    R361_2_O_RB_이상_리셋 AT %MW94020.10 : BOOL; (* R361_2_O_RB_이상_리셋 *)
    R361_2_O_RB_작업완료_리셋 AT %MW94020.8 : BOOL; (* R361_2_O_RB_작업완료_리셋 *)
    R363_1_I_RB_0_5_COMM_CHK AT %MW84033.14 : BOOL; (* R363_1_I_RB_0_5_COMM_CHK *)
    R363_1_I_RB_10차_간섭무 AT %MW84031.9 : BOOL; (* R363_1_I_RB_10차_간섭무 *)
    R363_1_I_RB_11차_간섭무 AT %MW84031.10 : BOOL; (* R363_1_I_RB_11차_간섭무 *)
    R363_1_I_RB_12차_간섭무 AT %MW84031.11 : BOOL; (* R363_1_I_RB_12차_간섭무 *)
    R363_1_I_RB_1차_간섭무 AT %MW84031.0 : BOOL; (* R363_1_I_RB_1차_간섭무 *)
    R363_1_I_RB_1차_작업완료 AT %MW84030.9 : BOOL; (* R363_1_I_RB_1차_작업완료 *)
    R363_1_I_RB_2차_간섭무 AT %MW84031.1 : BOOL; (* R363_1_I_RB_2차_간섭무 *)
    R363_1_I_RB_2차_작업완료 AT %MW84030.10 : BOOL; (* R363_1_I_RB_2차_작업완료 *)
    R363_1_I_RB_3차_간섭무 AT %MW84031.2 : BOOL; (* R363_1_I_RB_3차_간섭무 *)
    R363_1_I_RB_3차_작업완료 AT %MW84030.11 : BOOL; (* R363_1_I_RB_3차_작업완료 *)
    R363_1_I_RB_4차_간섭무 AT %MW84031.3 : BOOL; (* R363_1_I_RB_4차_간섭무 *)
    R363_1_I_RB_4차_작업완료 AT %MW84030.12 : BOOL; (* R363_1_I_RB_4차_작업완료 *)
    R363_1_I_RB_5차_간섭무 AT %MW84031.4 : BOOL; (* R363_1_I_RB_5차_간섭무 *)
    R363_1_I_RB_5차_작업완료 AT %MW84030.13 : BOOL; (* R363_1_I_RB_5차_작업완료 *)
    R363_1_I_RB_6차_간섭무 AT %MW84031.5 : BOOL; (* R363_1_I_RB_6차_간섭무 *)
    R363_1_I_RB_6차_작업완료 AT %MW84030.14 : BOOL; (* R363_1_I_RB_6차_작업완료 *)
    R363_1_I_RB_7차_간섭무 AT %MW84031.6 : BOOL; (* R363_1_I_RB_7차_간섭무 *)
    R363_1_I_RB_7차_작업완료 AT %MW84030.15 : BOOL; (* R363_1_I_RB_7차_작업완료 *)
    R363_1_I_RB_8차_간섭무 AT %MW84031.7 : BOOL; (* R363_1_I_RB_8차_간섭무 *)
    R363_1_I_RB_9차_간섭무 AT %MW84031.8 : BOOL; (* R363_1_I_RB_9차_간섭무 *)
    R363_1_I_RB_AB_NORMAL_선택 AT %MW84030.6 : BOOL; (* R363_1_I_RB_AB_NORMAL_선택 *)
    R363_1_I_RB_GUN1_FIXED_TIP AT %MW84037 : WORD; (* R363_1_I_RB_GUN1_FIXED_TIP *)
    R363_1_I_RB_GUN1_MOVING_TIP AT %MW84036 : WORD; (* R363_1_I_RB_GUN1_MOVING_TIP *)
    R363_1_I_RB_GUN2_FIXED_TIP AT %MW84039 : WORD; (* R363_1_I_RB_GUN2_FIXED_TIP *)
    R363_1_I_RB_GUN2_MOVING_TIP AT %MW84038 : WORD; (* R363_1_I_RB_GUN2_MOVING_TIP *)
    R363_1_I_RB_INPUT AT %MW84030 : ARRAY[0..3] OF WORD; (* R363_1_I_RB_INPUT *)
    R363_1_I_RB_LS_이상 AT %MW84032.11 : BOOL; (* R363_1_I_RB_LS_이상 *)
    R363_1_I_RB_MOTOR_MC_ON AT %MW84033.15 : BOOL; (* R363_1_I_RB_MOTOR_MC_ON *)
    R363_1_I_RB_PLT_UNLOAD_완료 AT %MW84033.11 : BOOL; (* R363_1_I_RB_PLT_UNLOAD_완료 *)
    R363_1_I_RB_PLT_최종UNLOAD_완료 AT %MW84033.12 : BOOL; (* R363_1_I_RB_PLT_최종UNLOAD_완료 *)
    R363_1_I_RB_PROG_ECHO_1 AT %MW84032.0 : BOOL; (* R363_1_I_RB_PROG_ECHO_1 *)
    R363_1_I_RB_PROG_ECHO_128 AT %MW84032.7 : BOOL; (* R363_1_I_RB_PROG_ECHO_128 *)
    R363_1_I_RB_PROG_ECHO_16 AT %MW84032.4 : BOOL; (* R363_1_I_RB_PROG_ECHO_16 *)
    R363_1_I_RB_PROG_ECHO_2 AT %MW84032.1 : BOOL; (* R363_1_I_RB_PROG_ECHO_2 *)
    R363_1_I_RB_PROG_ECHO_32 AT %MW84032.5 : BOOL; (* R363_1_I_RB_PROG_ECHO_32 *)
    R363_1_I_RB_PROG_ECHO_4 AT %MW84032.2 : BOOL; (* R363_1_I_RB_PROG_ECHO_4 *)
    R363_1_I_RB_PROG_ECHO_64 AT %MW84032.6 : BOOL; (* R363_1_I_RB_PROG_ECHO_64 *)
    R363_1_I_RB_PROG_ECHO_8 AT %MW84032.3 : BOOL; (* R363_1_I_RB_PROG_ECHO_8 *)
    R363_1_I_RB_SP3_8 AT %MW84033.8 : BOOL; (* R363_1_I_RB_SP3_8 *)
    R363_1_I_RB_SP3_9 AT %MW84033.9 : BOOL; (* R363_1_I_RB_SP3_9 *)
    R363_1_I_RB_SPARE_WORD_4 AT %MW84034 : WORD; (* R363_1_I_RB_SPARE_WORD_4 *)
    R363_1_I_RB_SP_1_12 AT %MW84031.12 : BOOL; (* R363_1_I_RB_SP_1_12 *)
    R363_1_I_RB_SP_1_13 AT %MW84031.13 : BOOL; (* R363_1_I_RB_SP_1_13 *)
    R363_1_I_RB_SP_1_14 AT %MW84031.14 : BOOL; (* R363_1_I_RB_SP_1_14 *)
    R363_1_I_RB_SP_1_15 AT %MW84031.15 : BOOL; (* R363_1_I_RB_SP_1_15 *)
    R363_1_I_RB_TC_이상 AT %MW84032.8 : BOOL; (* R363_1_I_RB_TC_이상 *)
    R363_1_I_RB_TIP_CHANGE AT %MW84033.13 : BOOL; (* R363_1_I_RB_TIP_CHANGE *)
    R363_1_I_RB_TIP_DRESSING AT %MW84030.7 : BOOL; (* R363_1_I_RB_TIP_DRESSING *)
    R363_1_I_RB__PLT_카운터리셋완료 AT %MW84033.10 : BOOL; (* R363_1_I_RB__PLT_카운터리셋완료 *)
    R363_1_I_RB_공기압_이상 AT %MW84032.9 : BOOL; (* R363_1_I_RB_공기압_이상 *)
    R363_1_I_RB_냉각수_이상 AT %MW84032.10 : BOOL; (* R363_1_I_RB_냉각수_이상 *)
    R363_1_I_RB_비상정지_NC AT %MW84030.8 : BOOL; (* R363_1_I_RB_비상정지_NC *)
    R363_1_I_RB_비전이상 AT %MW84032.14 : BOOL; (* R363_1_I_RB_비전이상 *)
    R363_1_I_RB_상호인터록_INT1 AT %MW84033.0 : BOOL; (* R363_1_I_RB_상호인터록_INT1 *)
    R363_1_I_RB_상호인터록_INT2 AT %MW84033.1 : BOOL; (* R363_1_I_RB_상호인터록_INT2 *)
    R363_1_I_RB_상호인터록_INT3 AT %MW84033.2 : BOOL; (* R363_1_I_RB_상호인터록_INT3 *)
    R363_1_I_RB_상호인터록_INT4 AT %MW84033.3 : BOOL; (* R363_1_I_RB_상호인터록_INT4 *)
    R363_1_I_RB_상호인터록_INT5 AT %MW84033.4 : BOOL; (* R363_1_I_RB_상호인터록_INT5 *)
    R363_1_I_RB_상호인터록_INT6 AT %MW84033.5 : BOOL; (* R363_1_I_RB_상호인터록_INT6 *)
    R363_1_I_RB_상호인터록_INT7 AT %MW84033.6 : BOOL; (* R363_1_I_RB_상호인터록_INT7 *)
    R363_1_I_RB_상호인터록_INT8 AT %MW84033.7 : BOOL; (* R363_1_I_RB_상호인터록_INT8 *)
    R363_1_I_RB_실러이상 AT %MW84032.13 : BOOL; (* R363_1_I_RB_실러이상 *)
    R363_1_I_RB_용접카운터이상 AT %MW84032.15 : BOOL; (* R363_1_I_RB_용접카운터이상 *)
    R363_1_I_RB_용접타점수 AT %MW84035 : WORD; (* R363_1_I_RB_용접타점수 *)
    R363_1_I_RB_운전준비 AT %MW84030.3 : BOOL; (* R363_1_I_RB_운전준비 *)
    R363_1_I_RB_원위치 AT %MW84030.0 : BOOL; (* R363_1_I_RB_원위치 *)
    R363_1_I_RB_이상리셋 AT %MW84030.2 : BOOL; (* R363_1_I_RB_이상리셋 *)
    R363_1_I_RB_자동 AT %MW84030.4 : BOOL; (* R363_1_I_RB_자동 *)
    R363_1_I_RB_자동기동 AT %MW84030.5 : BOOL; (* R363_1_I_RB_자동기동 *)
    R363_1_I_RB_최종_작업완료 AT %MW84030.1 : BOOL; (* R363_1_I_RB_최종_작업완료 *)
    R363_1_I_RB_통신이상 AT %MW84032.12 : BOOL; (* R363_1_I_RB_통신이상 *)
    R363_1_M_I_RB_1차_작업완료 AT %MW20031.2 : BOOL; (* R363_1_M_I_RB_1차_작업완료 *)
    R363_1_M_I_RB_2차_작업완료 AT %MW20031.3 : BOOL; (* R363_1_M_I_RB_2차_작업완료 *)
    R363_1_M_I_RB_3차_작업완료 AT %MW20031.4 : BOOL; (* R363_1_M_I_RB_3차_작업완료 *)
    R363_1_M_I_RB_4차_작업완료 AT %MW20031.5 : BOOL; (* R363_1_M_I_RB_4차_작업완료 *)
    R363_1_M_I_RB_5차_작업완료 AT %MW20031.6 : BOOL; (* R363_1_M_I_RB_5차_작업완료 *)
    R363_1_M_I_RB_6차_작업완료 AT %MW20031.7 : BOOL; (* R363_1_M_I_RB_6차_작업완료 *)
    R363_1_M_I_RB_7차_작업완료 AT %MW20031.8 : BOOL; (* R363_1_M_I_RB_7차_작업완료 *)
    R363_1_M_I_RB_PAUSE_보조 AT %MW20030.5 : BOOL; (* R363_1_M_I_RB_PAUSE_보조 *)
    R363_1_M_I_RB_PLC_RUN_CHK_이상 AT %MW20030.7 : BOOL; (* R363_1_M_I_RB_PLC_RUN_CHK_이상 *)
    R363_1_M_I_RB_간섭무_1 AT %MW20032.0 : BOOL; (* R363_1_M_I_RB_간섭무_1 *)
    R363_1_M_I_RB_간섭무_10 AT %MW20032.9 : BOOL; (* R363_1_M_I_RB_간섭무_10 *)
    R363_1_M_I_RB_간섭무_11 AT %MW20032.10 : BOOL; (* R363_1_M_I_RB_간섭무_11 *)
    R363_1_M_I_RB_간섭무_12 AT %MW20032.11 : BOOL; (* R363_1_M_I_RB_간섭무_12 *)
    R363_1_M_I_RB_간섭무_2 AT %MW20032.1 : BOOL; (* R363_1_M_I_RB_간섭무_2 *)
    R363_1_M_I_RB_간섭무_3 AT %MW20032.2 : BOOL; (* R363_1_M_I_RB_간섭무_3 *)
    R363_1_M_I_RB_간섭무_4 AT %MW20032.3 : BOOL; (* R363_1_M_I_RB_간섭무_4 *)
    R363_1_M_I_RB_간섭무_5 AT %MW20032.4 : BOOL; (* R363_1_M_I_RB_간섭무_5 *)
    R363_1_M_I_RB_간섭무_6 AT %MW20032.5 : BOOL; (* R363_1_M_I_RB_간섭무_6 *)
    R363_1_M_I_RB_간섭무_7 AT %MW20032.6 : BOOL; (* R363_1_M_I_RB_간섭무_7 *)
    R363_1_M_I_RB_간섭무_8 AT %MW20032.7 : BOOL; (* R363_1_M_I_RB_간섭무_8 *)
    R363_1_M_I_RB_간섭무_9 AT %MW20032.8 : BOOL; (* R363_1_M_I_RB_간섭무_9 *)
    R363_1_M_I_RB_비상정지 AT %MW20030.4 : BOOL; (* R363_1_M_I_RB_비상정지 *)
    R363_1_M_I_RB_운전준비 AT %MW20030.0 : BOOL; (* R363_1_M_I_RB_운전준비 *)
    R363_1_M_I_RB_원위치 AT %MW20030.3 : BOOL; (* R363_1_M_I_RB_원위치 *)
    R363_1_M_I_RB_이상 AT %MW20030.2 : BOOL; (* R363_1_M_I_RB_이상 *)
    R363_1_M_I_RB_자동 AT %MW20030.1 : BOOL; (* R363_1_M_I_RB_자동 *)
    R363_1_M_I_RB_최종작업완료 AT %MW20031.0 : BOOL; (* R363_1_M_I_RB_최종작업완료 *)
    R363_1_M_I_RB_프로그램_이상 AT %MW20030.6 : BOOL; (* R363_1_M_I_RB_프로그램_이상 *)
    R363_1_M_O_RB_1_CYCLE_SET AT %MW21030.3 : BOOL; (* R363_1_M_O_RB_1_CYCLE_SET *)
    R363_1_M_O_RB_1_CYCLE_리셋 AT %MW21030.4 : BOOL; (* R363_1_M_O_RB_1_CYCLE_리셋 *)
    R363_1_M_O_RB_1차_작업완료_리셋 AT %MW21032.0 : BOOL; (* R363_1_M_O_RB_1차_작업완료_리셋 *)
    R363_1_M_O_RB_2차_작업완료_리셋 AT %MW21032.1 : BOOL; (* R363_1_M_O_RB_2차_작업완료_리셋 *)
    R363_1_M_O_RB_2차_진입OK AT %MW21031.8 : BOOL; (* R363_1_M_O_RB_2차_진입OK *)
    R363_1_M_O_RB_3차_작업완료_리셋 AT %MW21032.2 : BOOL; (* R363_1_M_O_RB_3차_작업완료_리셋 *)
    R363_1_M_O_RB_3차_진입OK AT %MW21031.9 : BOOL; (* R363_1_M_O_RB_3차_진입OK *)
    R363_1_M_O_RB_4차_작업완료_리셋 AT %MW21032.3 : BOOL; (* R363_1_M_O_RB_4차_작업완료_리셋 *)
    R363_1_M_O_RB_4차_진입OK AT %MW21031.10 : BOOL; (* R363_1_M_O_RB_4차_진입OK *)
    R363_1_M_O_RB_5차_작업완료_리셋 AT %MW21032.4 : BOOL; (* R363_1_M_O_RB_5차_작업완료_리셋 *)
    R363_1_M_O_RB_5차_진입OK AT %MW21031.11 : BOOL; (* R363_1_M_O_RB_5차_진입OK *)
    R363_1_M_O_RB_6차_작업완료_리셋 AT %MW21032.5 : BOOL; (* R363_1_M_O_RB_6차_작업완료_리셋 *)
    R363_1_M_O_RB_6차_진입OK AT %MW21031.12 : BOOL; (* R363_1_M_O_RB_6차_진입OK *)
    R363_1_M_O_RB_7차_작업완료_리셋 AT %MW21032.6 : BOOL; (* R363_1_M_O_RB_7차_작업완료_리셋 *)
    R363_1_M_O_RB_7차_진입OK AT %MW21031.13 : BOOL; (* R363_1_M_O_RB_7차_진입OK *)
    R363_1_M_O_RB_ATD_OK AT %MW21030.6 : BOOL; (* R363_1_M_O_RB_ATD_OK *)
    R363_1_M_O_RB_PLT_10_진입OK AT %MW21033.10 : BOOL; (* R363_1_M_O_RB_PLT_10_진입OK *)
    R363_1_M_O_RB_PLT_11_진입OK AT %MW21033.11 : BOOL; (* R363_1_M_O_RB_PLT_11_진입OK *)
    R363_1_M_O_RB_PLT_12_진입OK AT %MW21033.12 : BOOL; (* R363_1_M_O_RB_PLT_12_진입OK *)
    R363_1_M_O_RB_PLT_1_진입OK AT %MW21033.1 : BOOL; (* R363_1_M_O_RB_PLT_1_진입OK *)
    R363_1_M_O_RB_PLT_2_진입OK AT %MW21033.2 : BOOL; (* R363_1_M_O_RB_PLT_2_진입OK *)
    R363_1_M_O_RB_PLT_3_진입OK AT %MW21033.3 : BOOL; (* R363_1_M_O_RB_PLT_3_진입OK *)
    R363_1_M_O_RB_PLT_4_진입OK AT %MW21033.4 : BOOL; (* R363_1_M_O_RB_PLT_4_진입OK *)
    R363_1_M_O_RB_PLT_5_진입OK AT %MW21033.5 : BOOL; (* R363_1_M_O_RB_PLT_5_진입OK *)
    R363_1_M_O_RB_PLT_6_진입OK AT %MW21033.6 : BOOL; (* R363_1_M_O_RB_PLT_6_진입OK *)
    R363_1_M_O_RB_PLT_7_진입OK AT %MW21033.7 : BOOL; (* R363_1_M_O_RB_PLT_7_진입OK *)
    R363_1_M_O_RB_PLT_8_진입OK AT %MW21033.8 : BOOL; (* R363_1_M_O_RB_PLT_8_진입OK *)
    R363_1_M_O_RB_PLT_9_진입OK AT %MW21033.9 : BOOL; (* R363_1_M_O_RB_PLT_9_진입OK *)
    R363_1_M_O_RB_PLT_카운터리셋_보조 AT %MW21030.10 : BOOL; (* R363_1_M_O_RB_PLT_카운터리셋_보조 *)
    R363_1_M_O_RB_PROG_NO AT %MW21034 : WORD;
    R363_1_M_O_RB_RESTART_OK AT %MW21030.2 : BOOL; (* R363_1_M_O_RB_RESTART_OK *)
    R363_1_M_O_RB_START_OK AT %MW21030.0 : BOOL; (* R363_1_M_O_RB_START_OK *)
    R363_1_M_O_RB_TEST_MODE_5000회 AT %MW21030.12 : BOOL; (* R363_1_M_O_RB_TEST_MODE_5000회 *)
    R363_1_M_O_RB_TIP_교체_시작 AT %MW21030.7 : BOOL; (* R363_1_M_O_RB_TIP_교체_시작 *)
    R363_1_M_O_RB_TIP_교체_완료 AT %MW21030.8 : BOOL; (* R363_1_M_O_RB_TIP_교체_완료 *)
    R363_1_M_O_RB_VIP_MODE AT %MW21030.11 : BOOL; (* R363_1_M_O_RB_VIP_MODE *)
    R363_1_M_O_RB_냉각수_차단_요청 AT %MW21030.9 : BOOL; (* R363_1_M_O_RB_냉각수_차단_요청 *)
    R363_1_M_O_RB_진입OK_AX차종 AT %MW21031.0 : BOOL; (* R363_1_M_O_RB_진입OK_AX차종 *)
    R363_1_M_O_RB_진입OK_B차종 AT %MW21031.1 : BOOL; (* R363_1_M_O_RB_진입OK_B차종 *)
    R363_1_M_O_RB_진입OK_C차종 AT %MW21031.2 : BOOL; (* R363_1_M_O_RB_진입OK_C차종 *)
    R363_1_M_O_RB_진입OK_D차종 AT %MW21031.3 : BOOL; (* R363_1_M_O_RB_진입OK_D차종 *)
    R363_1_M_O_RB_진입OK_E차종 AT %MW21031.4 : BOOL; (* R363_1_M_O_RB_진입OK_E차종 *)
    R363_1_M_O_RB_진입OK_F차종 AT %MW21031.5 : BOOL; (* R363_1_M_O_RB_진입OK_F차종 *)
    R363_1_M_O_RB_진입OK_G차종 AT %MW21031.6 : BOOL; (* R363_1_M_O_RB_진입OK_G차종 *)
    R363_1_M_O_RB_진입OK_H차종 AT %MW21031.7 : BOOL; (* R363_1_M_O_RB_진입OK_H차종 *)
    R363_1_M_O_RB_최종_작업완료_리셋 AT %MW21030.5 : BOOL; (* R363_1_M_O_RB_최종_작업완료_리셋 *)
    R363_1_M_O_RB_프로그램_OK AT %MW21030.1 : BOOL; (* R363_1_M_O_RB_프로그램_OK *)
    R363_1_O_RB_0_5S_통신_CHK AT %MW94033.14 : BOOL; (* R363_1_O_RB_0_5S_통신_CHK *)
    R363_1_O_RB_2차_진입OK AT %MW94031.8 : BOOL; (* R363_1_O_RB_2차_진입OK *)
    R363_1_O_RB_3차_진입OK AT %MW94031.9 : BOOL; (* R363_1_O_RB_3차_진입OK *)
    R363_1_O_RB_4차_진입OK AT %MW94031.10 : BOOL; (* R363_1_O_RB_4차_진입OK *)
    R363_1_O_RB_5차_진입OK AT %MW94031.11 : BOOL; (* R363_1_O_RB_5차_진입OK *)
    R363_1_O_RB_6차_진입OK AT %MW94031.12 : BOOL; (* R363_1_O_RB_6차_진입OK *)
    R363_1_O_RB_7차_진입OK AT %MW94031.13 : BOOL; (* R363_1_O_RB_7차_진입OK *)
    R363_1_O_RB_AX_1차_진입OK AT %MW94031.0 : BOOL; (* R363_1_O_RB_AX_1차_진입OK *)
    R363_1_O_RB_B_1차_진입OK AT %MW94031.1 : BOOL; (* R363_1_O_RB_B_1차_진입OK *)
    R363_1_O_RB_C_1차_진입OK AT %MW94031.2 : BOOL; (* R363_1_O_RB_C_1차_진입OK *)
    R363_1_O_RB_D_1차_진입OK AT %MW94031.3 : BOOL; (* R363_1_O_RB_D_1차_진입OK *)
    R363_1_O_RB_EACH_작업완료_리셋 AT %MW94030.14 : BOOL; (* R363_1_O_RB_EACH_작업완료_리셋 *)
    R363_1_O_RB_EXT_READY AT %MW94030.11 : BOOL; (* R363_1_O_RB_EXT_READY *)
    R363_1_O_RB_E_1차_진입OK AT %MW94031.4 : BOOL; (* R363_1_O_RB_E_1차_진입OK *)
    R363_1_O_RB_F_1차_진입OK AT %MW94031.5 : BOOL; (* R363_1_O_RB_F_1차_진입OK *)
    R363_1_O_RB_GATE_OPEN_NC AT %MW94033.11 : BOOL; (* R363_1_O_RB_GATE_OPEN_NC *)
    R363_1_O_RB_G_1차_진입OK AT %MW94031.6 : BOOL; (* R363_1_O_RB_G_1차_진입OK *)
    R363_1_O_RB_H_1차_진입OK AT %MW94031.7 : BOOL; (* R363_1_O_RB_H_1차_진입OK *)
    R363_1_O_RB_OUTPUT AT %MW94030 : ARRAY[0..3] OF WORD; (* R363_1_O_RB_OUTPUT *)
    R363_1_O_RB_PAUSE_NC AT %MW94030.13 : BOOL; (* R363_1_O_RB_PAUSE_NC *)
    R363_1_O_RB_PLT10_진입OK AT %MW94032.9 : BOOL; (* R363_1_O_RB_PLT10_진입OK *)
    R363_1_O_RB_PLT11_진입OK AT %MW94032.10 : BOOL; (* R363_1_O_RB_PLT11_진입OK *)
    R363_1_O_RB_PLT12_진입OK AT %MW94032.11 : BOOL; (* R363_1_O_RB_PLT12_진입OK *)
    R363_1_O_RB_PLT1_진입OK AT %MW94032.0 : BOOL; (* R363_1_O_RB_PLT1_진입OK *)
    R363_1_O_RB_PLT2_진입OK AT %MW94032.1 : BOOL; (* R363_1_O_RB_PLT2_진입OK *)
    R363_1_O_RB_PLT3_진입OK AT %MW94032.2 : BOOL; (* R363_1_O_RB_PLT3_진입OK *)
    R363_1_O_RB_PLT4_진입OK AT %MW94032.3 : BOOL; (* R363_1_O_RB_PLT4_진입OK *)
    R363_1_O_RB_PLT5_진입OK AT %MW94032.4 : BOOL; (* R363_1_O_RB_PLT5_진입OK *)
    R363_1_O_RB_PLT6_진입OK AT %MW94032.5 : BOOL; (* R363_1_O_RB_PLT6_진입OK *)
    R363_1_O_RB_PLT7_진입OK AT %MW94032.6 : BOOL; (* R363_1_O_RB_PLT7_진입OK *)
    R363_1_O_RB_PLT8_진입OK AT %MW94032.7 : BOOL; (* R363_1_O_RB_PLT8_진입OK *)
    R363_1_O_RB_PLT9_진입OK AT %MW94032.8 : BOOL; (* R363_1_O_RB_PLT9_진입OK *)
    R363_1_O_RB_PLT_카운터_리셋_요구 AT %MW94033.10 : BOOL; (* R363_1_O_RB_PLT_카운터_리셋_요구 *)
    R363_1_O_RB_PROG_선택1 AT %MW94030.0 : BOOL; (* R363_1_O_RB_PROG_선택1 *)
    R363_1_O_RB_PROG_선택128 AT %MW94030.7 : BOOL; (* R363_1_O_RB_PROG_선택128 *)
    R363_1_O_RB_PROG_선택16 AT %MW94030.4 : BOOL; (* R363_1_O_RB_PROG_선택16 *)
    R363_1_O_RB_PROG_선택2 AT %MW94030.1 : BOOL; (* R363_1_O_RB_PROG_선택2 *)
    R363_1_O_RB_PROG_선택32 AT %MW94030.5 : BOOL; (* R363_1_O_RB_PROG_선택32 *)
    R363_1_O_RB_PROG_선택4 AT %MW94030.2 : BOOL; (* R363_1_O_RB_PROG_선택4 *)
    R363_1_O_RB_PROG_선택64 AT %MW94030.6 : BOOL; (* R363_1_O_RB_PROG_선택64 *)
    R363_1_O_RB_PROG_선택8 AT %MW94030.3 : BOOL; (* R363_1_O_RB_PROG_선택8 *)
    R363_1_O_RB_SP_1_14 AT %MW94031.14 : BOOL; (* R363_1_O_RB_SP_1_14 *)
    R363_1_O_RB_SP_1_15 AT %MW94031.15 : BOOL; (* R363_1_O_RB_SP_1_15 *)
    R363_1_O_RB_SP_2_12 AT %MW94032.12 : BOOL; (* R363_1_O_RB_SP_2_12 *)
    R363_1_O_RB_SP_2_13 AT %MW94032.13 : BOOL; (* R363_1_O_RB_SP_2_13 *)
    R363_1_O_RB_SP_2_14 AT %MW94032.14 : BOOL; (* R363_1_O_RB_SP_2_14 *)
    R363_1_O_RB_SP_5000TH_ON AT %MW94032.15 : BOOL; (* R363_1_O_RB_SP_5000TH_ON *)
    R363_1_O_RB_TIP_CHANGE_END AT %MW94033.9 : BOOL; (* R363_1_O_RB_TIP_CHANGE_END *)
    R363_1_O_RB_TIP_CHANGE_START AT %MW94033.8 : BOOL; (* R363_1_O_RB_TIP_CHANGE_START *)
    R363_1_O_RB_TIP_DRESS_SATRT AT %MW94030.12 : BOOL; (* R363_1_O_RB_TIP_DRESS_SATRT *)
    R363_1_O_RB_VIP_MODE AT %MW94033.15 : BOOL; (* R363_1_O_RB_VIP_MODE *)
    R363_1_O_RB_기동 AT %MW94030.9 : BOOL; (* R363_1_O_RB_기동 *)
    R363_1_O_RB_냉각수차단 AT %MW94030.15 : BOOL; (* R363_1_O_RB_냉각수차단 *)
    R363_1_O_RB_부저정지 AT %MW94033.13 : BOOL; (* R363_1_O_RB_부저정지 *)
    R363_1_O_RB_비상정지_NC AT %MW94033.12 : BOOL; (* R363_1_O_RB_비상정지_NC *)
    R363_1_O_RB_상호인터록_INT1 AT %MW94033.0 : BOOL; (* R363_1_O_RB_상호인터록_INT1 *)
    R363_1_O_RB_상호인터록_INT2 AT %MW94033.1 : BOOL; (* R363_1_O_RB_상호인터록_INT2 *)
    R363_1_O_RB_상호인터록_INT3 AT %MW94033.2 : BOOL; (* R363_1_O_RB_상호인터록_INT3 *)
    R363_1_O_RB_상호인터록_INT4 AT %MW94033.3 : BOOL; (* R363_1_O_RB_상호인터록_INT4 *)
    R363_1_O_RB_상호인터록_INT5 AT %MW94033.4 : BOOL; (* R363_1_O_RB_상호인터록_INT5 *)
    R363_1_O_RB_상호인터록_INT6 AT %MW94033.5 : BOOL; (* R363_1_O_RB_상호인터록_INT6 *)
    R363_1_O_RB_상호인터록_INT7 AT %MW94033.6 : BOOL; (* R363_1_O_RB_상호인터록_INT7 *)
    R363_1_O_RB_상호인터록_INT8 AT %MW94033.7 : BOOL; (* R363_1_O_RB_상호인터록_INT8 *)
    R363_1_O_RB_이상_리셋 AT %MW94030.10 : BOOL; (* R363_1_O_RB_이상_리셋 *)
    R363_1_O_RB_작업완료_리셋 AT %MW94030.8 : BOOL; (* R363_1_O_RB_작업완료_리셋 *)
    R363_2_I_RB_0_5_COMM_CHK AT %MW84043.14 : BOOL; (* R363_2_I_RB_0_5_COMM_CHK *)
    R363_2_I_RB_10차_간섭무 AT %MW84041.9 : BOOL; (* R363_2_I_RB_10차_간섭무 *)
    R363_2_I_RB_11차_간섭무 AT %MW84041.10 : BOOL; (* R363_2_I_RB_11차_간섭무 *)
    R363_2_I_RB_12차_간섭무 AT %MW84041.11 : BOOL; (* R363_2_I_RB_12차_간섭무 *)
    R363_2_I_RB_1차_간섭무 AT %MW84041.0 : BOOL; (* R363_2_I_RB_1차_간섭무 *)
    R363_2_I_RB_1차_작업완료 AT %MW84040.9 : BOOL; (* R363_2_I_RB_1차_작업완료 *)
    R363_2_I_RB_2차_간섭무 AT %MW84041.1 : BOOL; (* R363_2_I_RB_2차_간섭무 *)
    R363_2_I_RB_2차_작업완료 AT %MW84040.10 : BOOL; (* R363_2_I_RB_2차_작업완료 *)
    R363_2_I_RB_3차_간섭무 AT %MW84041.2 : BOOL; (* R363_2_I_RB_3차_간섭무 *)
    R363_2_I_RB_3차_작업완료 AT %MW84040.11 : BOOL; (* R363_2_I_RB_3차_작업완료 *)
    R363_2_I_RB_4차_간섭무 AT %MW84041.3 : BOOL; (* R363_2_I_RB_4차_간섭무 *)
    R363_2_I_RB_4차_작업완료 AT %MW84040.12 : BOOL; (* R363_2_I_RB_4차_작업완료 *)
    R363_2_I_RB_5차_간섭무 AT %MW84041.4 : BOOL; (* R363_2_I_RB_5차_간섭무 *)
    R363_2_I_RB_5차_작업완료 AT %MW84040.13 : BOOL; (* R363_2_I_RB_5차_작업완료 *)
    R363_2_I_RB_6차_간섭무 AT %MW84041.5 : BOOL; (* R363_2_I_RB_6차_간섭무 *)
    R363_2_I_RB_6차_작업완료 AT %MW84040.14 : BOOL; (* R363_2_I_RB_6차_작업완료 *)
    R363_2_I_RB_7차_간섭무 AT %MW84041.6 : BOOL; (* R363_2_I_RB_7차_간섭무 *)
    R363_2_I_RB_7차_작업완료 AT %MW84040.15 : BOOL; (* R363_2_I_RB_7차_작업완료 *)
    R363_2_I_RB_8차_간섭무 AT %MW84041.7 : BOOL; (* R363_2_I_RB_8차_간섭무 *)
    R363_2_I_RB_9차_간섭무 AT %MW84041.8 : BOOL; (* R363_2_I_RB_9차_간섭무 *)
    R363_2_I_RB_AB_NORMAL_선택 AT %MW84040.6 : BOOL; (* R363_2_I_RB_AB_NORMAL_선택 *)
    R363_2_I_RB_GUN1_FIXED_TIP AT %MW84047 : WORD; (* R363_2_I_RB_GUN1_FIXED_TIP *)
    R363_2_I_RB_GUN1_MOVING_TIP AT %MW84046 : WORD; (* R363_2_I_RB_GUN1_MOVING_TIP *)
    R363_2_I_RB_GUN2_FIXED_TIP AT %MW84049 : WORD; (* R363_2_I_RB_GUN2_FIXED_TIP *)
    R363_2_I_RB_GUN2_MOVING_TIP AT %MW84048 : WORD; (* R363_2_I_RB_GUN2_MOVING_TIP *)
    R363_2_I_RB_INPUT AT %MW84040 : ARRAY[0..3] OF WORD; (* R363_2_I_RB_INPUT *)
    R363_2_I_RB_LS_이상 AT %MW84042.11 : BOOL; (* R363_2_I_RB_LS_이상 *)
    R363_2_I_RB_MOTOR_MC_ON AT %MW84043.15 : BOOL; (* R363_2_I_RB_MOTOR_MC_ON *)
    R363_2_I_RB_PLT_UNLOAD_완료 AT %MW84043.11 : BOOL; (* R363_2_I_RB_PLT_UNLOAD_완료 *)
    R363_2_I_RB_PLT_최종UNLOAD_완료 AT %MW84043.12 : BOOL; (* R363_2_I_RB_PLT_최종UNLOAD_완료 *)
    R363_2_I_RB_PROG_ECHO_1 AT %MW84042.0 : BOOL; (* R363_2_I_RB_PROG_ECHO_1 *)
    R363_2_I_RB_PROG_ECHO_128 AT %MW84042.7 : BOOL; (* R363_2_I_RB_PROG_ECHO_128 *)
    R363_2_I_RB_PROG_ECHO_16 AT %MW84042.4 : BOOL; (* R363_2_I_RB_PROG_ECHO_16 *)
    R363_2_I_RB_PROG_ECHO_2 AT %MW84042.1 : BOOL; (* R363_2_I_RB_PROG_ECHO_2 *)
    R363_2_I_RB_PROG_ECHO_32 AT %MW84042.5 : BOOL; (* R363_2_I_RB_PROG_ECHO_32 *)
    R363_2_I_RB_PROG_ECHO_4 AT %MW84042.2 : BOOL; (* R363_2_I_RB_PROG_ECHO_4 *)
    R363_2_I_RB_PROG_ECHO_64 AT %MW84042.6 : BOOL; (* R363_2_I_RB_PROG_ECHO_64 *)
    R363_2_I_RB_PROG_ECHO_8 AT %MW84042.3 : BOOL; (* R363_2_I_RB_PROG_ECHO_8 *)
    R363_2_I_RB_SP3_8 AT %MW84043.8 : BOOL; (* R363_2_I_RB_SP3_8 *)
    R363_2_I_RB_SP3_9 AT %MW84043.9 : BOOL; (* R363_2_I_RB_SP3_9 *)
    R363_2_I_RB_SPARE_WORD_4 AT %MW84044 : WORD; (* R363_2_I_RB_SPARE_WORD_4 *)
    R363_2_I_RB_SP_1_12 AT %MW84041.12 : BOOL; (* R363_2_I_RB_SP_1_12 *)
    R363_2_I_RB_SP_1_13 AT %MW84041.13 : BOOL; (* R363_2_I_RB_SP_1_13 *)
    R363_2_I_RB_SP_1_14 AT %MW84041.14 : BOOL; (* R363_2_I_RB_SP_1_14 *)
    R363_2_I_RB_SP_1_15 AT %MW84041.15 : BOOL; (* R363_2_I_RB_SP_1_15 *)
    R363_2_I_RB_TC_이상 AT %MW84042.8 : BOOL; (* R363_2_I_RB_TC_이상 *)
    R363_2_I_RB_TIP_CHANGE AT %MW84043.13 : BOOL; (* R363_2_I_RB_TIP_CHANGE *)
    R363_2_I_RB_TIP_DRESSING AT %MW84040.7 : BOOL; (* R363_2_I_RB_TIP_DRESSING *)
    R363_2_I_RB__PLT_카운터리셋완료 AT %MW84043.10 : BOOL; (* R363_2_I_RB__PLT_카운터리셋완료 *)
    R363_2_I_RB_공기압_이상 AT %MW84042.9 : BOOL; (* R363_2_I_RB_공기압_이상 *)
    R363_2_I_RB_냉각수_이상 AT %MW84042.10 : BOOL; (* R363_2_I_RB_냉각수_이상 *)
    R363_2_I_RB_비상정지_NC AT %MW84040.8 : BOOL; (* R363_2_I_RB_비상정지_NC *)
    R363_2_I_RB_비전이상 AT %MW84042.14 : BOOL; (* R363_2_I_RB_비전이상 *)
    R363_2_I_RB_상호인터록_INT1 AT %MW84043.0 : BOOL; (* R363_2_I_RB_상호인터록_INT1 *)
    R363_2_I_RB_상호인터록_INT2 AT %MW84043.1 : BOOL; (* R363_2_I_RB_상호인터록_INT2 *)
    R363_2_I_RB_상호인터록_INT3 AT %MW84043.2 : BOOL; (* R363_2_I_RB_상호인터록_INT3 *)
    R363_2_I_RB_상호인터록_INT4 AT %MW84043.3 : BOOL; (* R363_2_I_RB_상호인터록_INT4 *)
    R363_2_I_RB_상호인터록_INT5 AT %MW84043.4 : BOOL; (* R363_2_I_RB_상호인터록_INT5 *)
    R363_2_I_RB_상호인터록_INT6 AT %MW84043.5 : BOOL; (* R363_2_I_RB_상호인터록_INT6 *)
    R363_2_I_RB_상호인터록_INT7 AT %MW84043.6 : BOOL; (* R363_2_I_RB_상호인터록_INT7 *)
    R363_2_I_RB_상호인터록_INT8 AT %MW84043.7 : BOOL; (* R363_2_I_RB_상호인터록_INT8 *)
    R363_2_I_RB_실러이상 AT %MW84042.13 : BOOL; (* R363_2_I_RB_실러이상 *)
    R363_2_I_RB_용접카운터이상 AT %MW84042.15 : BOOL; (* R363_2_I_RB_용접카운터이상 *)
    R363_2_I_RB_용접타점수 AT %MW84045 : WORD; (* R363_2_I_RB_용접타점수 *)
    R363_2_I_RB_운전준비 AT %MW84040.3 : BOOL; (* R363_2_I_RB_운전준비 *)
    R363_2_I_RB_원위치 AT %MW84040.0 : BOOL; (* R363_2_I_RB_원위치 *)
    R363_2_I_RB_이상리셋 AT %MW84040.2 : BOOL; (* R363_2_I_RB_이상리셋 *)
    R363_2_I_RB_자동 AT %MW84040.4 : BOOL; (* R363_2_I_RB_자동 *)
    R363_2_I_RB_자동기동 AT %MW84040.5 : BOOL; (* R363_2_I_RB_자동기동 *)
    R363_2_I_RB_최종_작업완료 AT %MW84040.1 : BOOL; (* R363_2_I_RB_최종_작업완료 *)
    R363_2_I_RB_통신이상 AT %MW84042.12 : BOOL; (* R363_2_I_RB_통신이상 *)
    R363_2_M_I_RB_1차_작업완료 AT %MW20041.2 : BOOL; (* R363_2_M_I_RB_1차_작업완료 *)
    R363_2_M_I_RB_2차_작업완료 AT %MW20041.3 : BOOL; (* R363_2_M_I_RB_2차_작업완료 *)
    R363_2_M_I_RB_3차_작업완료 AT %MW20041.4 : BOOL; (* R363_2_M_I_RB_3차_작업완료 *)
    R363_2_M_I_RB_4차_작업완료 AT %MW20041.5 : BOOL; (* R363_2_M_I_RB_4차_작업완료 *)
    R363_2_M_I_RB_5차_작업완료 AT %MW20041.6 : BOOL; (* R363_2_M_I_RB_5차_작업완료 *)
    R363_2_M_I_RB_6차_작업완료 AT %MW20041.7 : BOOL; (* R363_2_M_I_RB_6차_작업완료 *)
    R363_2_M_I_RB_7차_작업완료 AT %MW20041.8 : BOOL; (* R363_2_M_I_RB_7차_작업완료 *)
    R363_2_M_I_RB_PAUSE_보조 AT %MW20040.5 : BOOL; (* R363_2_M_I_RB_PAUSE_보조 *)
    R363_2_M_I_RB_PLC_RUN_CHK_이상 AT %MW20040.7 : BOOL; (* R363_2_M_I_RB_PLC_RUN_CHK_이상 *)
    R363_2_M_I_RB_간섭무_1 AT %MW20042.0 : BOOL; (* R363_2_M_I_RB_간섭무_1 *)
    R363_2_M_I_RB_간섭무_10 AT %MW20042.9 : BOOL; (* R363_2_M_I_RB_간섭무_10 *)
    R363_2_M_I_RB_간섭무_11 AT %MW20042.10 : BOOL; (* R363_2_M_I_RB_간섭무_11 *)
    R363_2_M_I_RB_간섭무_12 AT %MW20042.11 : BOOL; (* R363_2_M_I_RB_간섭무_12 *)
    R363_2_M_I_RB_간섭무_2 AT %MW20042.1 : BOOL; (* R363_2_M_I_RB_간섭무_2 *)
    R363_2_M_I_RB_간섭무_3 AT %MW20042.2 : BOOL; (* R363_2_M_I_RB_간섭무_3 *)
    R363_2_M_I_RB_간섭무_4 AT %MW20042.3 : BOOL; (* R363_2_M_I_RB_간섭무_4 *)
    R363_2_M_I_RB_간섭무_5 AT %MW20042.4 : BOOL; (* R363_2_M_I_RB_간섭무_5 *)
    R363_2_M_I_RB_간섭무_6 AT %MW20042.5 : BOOL; (* R363_2_M_I_RB_간섭무_6 *)
    R363_2_M_I_RB_간섭무_7 AT %MW20042.6 : BOOL; (* R363_2_M_I_RB_간섭무_7 *)
    R363_2_M_I_RB_간섭무_8 AT %MW20042.7 : BOOL; (* R363_2_M_I_RB_간섭무_8 *)
    R363_2_M_I_RB_간섭무_9 AT %MW20042.8 : BOOL; (* R363_2_M_I_RB_간섭무_9 *)
    R363_2_M_I_RB_비상정지 AT %MW20040.4 : BOOL; (* R363_2_M_I_RB_비상정지 *)
    R363_2_M_I_RB_운전준비 AT %MW20040.0 : BOOL; (* R363_2_M_I_RB_운전준비 *)
    R363_2_M_I_RB_원위치 AT %MW20040.3 : BOOL; (* R363_2_M_I_RB_원위치 *)
    R363_2_M_I_RB_이상 AT %MW20040.2 : BOOL; (* R363_2_M_I_RB_이상 *)
    R363_2_M_I_RB_자동 AT %MW20040.1 : BOOL; (* R363_2_M_I_RB_자동 *)
    R363_2_M_I_RB_최종작업완료 AT %MW20041.0 : BOOL; (* R363_2_M_I_RB_최종작업완료 *)
    R363_2_M_I_RB_프로그램_이상 AT %MW20040.6 : BOOL; (* R363_2_M_I_RB_프로그램_이상 *)
    R363_2_M_O_RB_1_CYCLE_SET AT %MW21040.3 : BOOL; (* R363_2_M_O_RB_1_CYCLE_SET *)
    R363_2_M_O_RB_1_CYCLE_리셋 AT %MW21040.4 : BOOL; (* R363_2_M_O_RB_1_CYCLE_리셋 *)
    R363_2_M_O_RB_1차_작업완료_리셋 AT %MW21042.0 : BOOL; (* R363_2_M_O_RB_1차_작업완료_리셋 *)
    R363_2_M_O_RB_2차_작업완료_리셋 AT %MW21042.1 : BOOL; (* R363_2_M_O_RB_2차_작업완료_리셋 *)
    R363_2_M_O_RB_2차_진입OK AT %MW21041.8 : BOOL; (* R363_2_M_O_RB_2차_진입OK *)
    R363_2_M_O_RB_3차_작업완료_리셋 AT %MW21042.2 : BOOL; (* R363_2_M_O_RB_3차_작업완료_리셋 *)
    R363_2_M_O_RB_3차_진입OK AT %MW21041.9 : BOOL; (* R363_2_M_O_RB_3차_진입OK *)
    R363_2_M_O_RB_4차_작업완료_리셋 AT %MW21042.3 : BOOL; (* R363_2_M_O_RB_4차_작업완료_리셋 *)
    R363_2_M_O_RB_4차_진입OK AT %MW21041.10 : BOOL; (* R363_2_M_O_RB_4차_진입OK *)
    R363_2_M_O_RB_5차_작업완료_리셋 AT %MW21042.4 : BOOL; (* R363_2_M_O_RB_5차_작업완료_리셋 *)
    R363_2_M_O_RB_5차_진입OK AT %MW21041.11 : BOOL; (* R363_2_M_O_RB_5차_진입OK *)
    R363_2_M_O_RB_6차_작업완료_리셋 AT %MW21042.5 : BOOL; (* R363_2_M_O_RB_6차_작업완료_리셋 *)
    R363_2_M_O_RB_6차_진입OK AT %MW21041.12 : BOOL; (* R363_2_M_O_RB_6차_진입OK *)
    R363_2_M_O_RB_7차_작업완료_리셋 AT %MW21042.6 : BOOL; (* R363_2_M_O_RB_7차_작업완료_리셋 *)
    R363_2_M_O_RB_7차_진입OK AT %MW21041.13 : BOOL; (* R363_2_M_O_RB_7차_진입OK *)
    R363_2_M_O_RB_ATD_OK AT %MW21040.6 : BOOL; (* R363_2_M_O_RB_ATD_OK *)
    R363_2_M_O_RB_PLT_10_진입OK AT %MW21043.10 : BOOL; (* R363_2_M_O_RB_PLT_10_진입OK *)
    R363_2_M_O_RB_PLT_11_진입OK AT %MW21043.11 : BOOL; (* R363_2_M_O_RB_PLT_11_진입OK *)
    R363_2_M_O_RB_PLT_12_진입OK AT %MW21043.12 : BOOL; (* R363_2_M_O_RB_PLT_12_진입OK *)
    R363_2_M_O_RB_PLT_1_진입OK AT %MW21043.1 : BOOL; (* R363_2_M_O_RB_PLT_1_진입OK *)
    R363_2_M_O_RB_PLT_2_진입OK AT %MW21043.2 : BOOL; (* R363_2_M_O_RB_PLT_2_진입OK *)
    R363_2_M_O_RB_PLT_3_진입OK AT %MW21043.3 : BOOL; (* R363_2_M_O_RB_PLT_3_진입OK *)
    R363_2_M_O_RB_PLT_4_진입OK AT %MW21043.4 : BOOL; (* R363_2_M_O_RB_PLT_4_진입OK *)
    R363_2_M_O_RB_PLT_5_진입OK AT %MW21043.5 : BOOL; (* R363_2_M_O_RB_PLT_5_진입OK *)
    R363_2_M_O_RB_PLT_6_진입OK AT %MW21043.6 : BOOL; (* R363_2_M_O_RB_PLT_6_진입OK *)
    R363_2_M_O_RB_PLT_7_진입OK AT %MW21043.7 : BOOL; (* R363_2_M_O_RB_PLT_7_진입OK *)
    R363_2_M_O_RB_PLT_8_진입OK AT %MW21043.8 : BOOL; (* R363_2_M_O_RB_PLT_8_진입OK *)
    R363_2_M_O_RB_PLT_9_진입OK AT %MW21043.9 : BOOL; (* R363_2_M_O_RB_PLT_9_진입OK *)
    R363_2_M_O_RB_PLT_카운터리셋_보조 AT %MW21040.10 : BOOL; (* R363_2_M_O_RB_PLT_카운터리셋_보조 *)
    R363_2_M_O_RB_PROG_NO AT %MW21044 : WORD;
    R363_2_M_O_RB_RESTART_OK AT %MW21040.2 : BOOL; (* R363_2_M_O_RB_RESTART_OK *)
    R363_2_M_O_RB_START_OK AT %MW21040.0 : BOOL; (* R363_2_M_O_RB_START_OK *)
    R363_2_M_O_RB_TEST_MODE_5000회 AT %MW21040.12 : BOOL; (* R363_2_M_O_RB_TEST_MODE_5000회 *)
    R363_2_M_O_RB_TIP_교체_시작 AT %MW21040.7 : BOOL; (* R363_2_M_O_RB_TIP_교체_시작 *)
    R363_2_M_O_RB_TIP_교체_완료 AT %MW21040.8 : BOOL; (* R363_2_M_O_RB_TIP_교체_완료 *)
    R363_2_M_O_RB_VIP_MODE AT %MW21040.11 : BOOL; (* R363_2_M_O_RB_VIP_MODE *)
    R363_2_M_O_RB_냉각수_차단_요청 AT %MW21040.9 : BOOL; (* R363_2_M_O_RB_냉각수_차단_요청 *)
    R363_2_M_O_RB_진입OK_AX차종 AT %MW21041.0 : BOOL; (* R363_2_M_O_RB_진입OK_AX차종 *)
    R363_2_M_O_RB_진입OK_B차종 AT %MW21041.1 : BOOL; (* R363_2_M_O_RB_진입OK_B차종 *)
    R363_2_M_O_RB_진입OK_C차종 AT %MW21041.2 : BOOL; (* R363_2_M_O_RB_진입OK_C차종 *)
    R363_2_M_O_RB_진입OK_D차종 AT %MW21041.3 : BOOL; (* R363_2_M_O_RB_진입OK_D차종 *)
    R363_2_M_O_RB_진입OK_E차종 AT %MW21041.4 : BOOL; (* R363_2_M_O_RB_진입OK_E차종 *)
    R363_2_M_O_RB_진입OK_F차종 AT %MW21041.5 : BOOL; (* R363_2_M_O_RB_진입OK_F차종 *)
    R363_2_M_O_RB_진입OK_G차종 AT %MW21041.6 : BOOL; (* R363_2_M_O_RB_진입OK_G차종 *)
    R363_2_M_O_RB_진입OK_H차종 AT %MW21041.7 : BOOL; (* R363_2_M_O_RB_진입OK_H차종 *)
    R363_2_M_O_RB_최종_작업완료_리셋 AT %MW21040.5 : BOOL; (* R363_2_M_O_RB_최종_작업완료_리셋 *)
    R363_2_M_O_RB_프로그램_OK AT %MW21040.1 : BOOL; (* R363_2_M_O_RB_프로그램_OK *)
    R363_2_O_RB_0_5S_통신_CHK AT %MW94043.14 : BOOL; (* R363_2_O_RB_0_5S_통신_CHK *)
    R363_2_O_RB_2차_진입OK AT %MW94041.8 : BOOL; (* R363_2_O_RB_2차_진입OK *)
    R363_2_O_RB_3차_진입OK AT %MW94041.9 : BOOL; (* R363_2_O_RB_3차_진입OK *)
    R363_2_O_RB_4차_진입OK AT %MW94041.10 : BOOL; (* R363_2_O_RB_4차_진입OK *)
    R363_2_O_RB_5차_진입OK AT %MW94041.11 : BOOL; (* R363_2_O_RB_5차_진입OK *)
    R363_2_O_RB_6차_진입OK AT %MW94041.12 : BOOL; (* R363_2_O_RB_6차_진입OK *)
    R363_2_O_RB_7차_진입OK AT %MW94041.13 : BOOL; (* R363_2_O_RB_7차_진입OK *)
    R363_2_O_RB_AX_1차_진입OK AT %MW94041.0 : BOOL; (* R363_2_O_RB_AX_1차_진입OK *)
    R363_2_O_RB_B_1차_진입OK AT %MW94041.1 : BOOL; (* R363_2_O_RB_B_1차_진입OK *)
    R363_2_O_RB_C_1차_진입OK AT %MW94041.2 : BOOL; (* R363_2_O_RB_C_1차_진입OK *)
    R363_2_O_RB_D_1차_진입OK AT %MW94041.3 : BOOL; (* R363_2_O_RB_D_1차_진입OK *)
    R363_2_O_RB_EACH_작업완료_리셋 AT %MW94040.14 : BOOL; (* R363_2_O_RB_EACH_작업완료_리셋 *)
    R363_2_O_RB_EXT_READY AT %MW94040.11 : BOOL; (* R363_2_O_RB_EXT_READY *)
    R363_2_O_RB_E_1차_진입OK AT %MW94041.4 : BOOL; (* R363_2_O_RB_E_1차_진입OK *)
    R363_2_O_RB_F_1차_진입OK AT %MW94041.5 : BOOL; (* R363_2_O_RB_F_1차_진입OK *)
    R363_2_O_RB_GATE_OPEN_NC AT %MW94043.11 : BOOL; (* R363_2_O_RB_GATE_OPEN_NC *)
    R363_2_O_RB_G_1차_진입OK AT %MW94041.6 : BOOL; (* R363_2_O_RB_G_1차_진입OK *)
    R363_2_O_RB_H_1차_진입OK AT %MW94041.7 : BOOL; (* R363_2_O_RB_H_1차_진입OK *)
    R363_2_O_RB_OUTPUT AT %MW94040 : ARRAY[0..3] OF WORD; (* R363_2_O_RB_OUTPUT *)
    R363_2_O_RB_PAUSE_NC AT %MW94040.13 : BOOL; (* R363_2_O_RB_PAUSE_NC *)
    R363_2_O_RB_PLT10_진입OK AT %MW94042.9 : BOOL; (* R363_2_O_RB_PLT10_진입OK *)
    R363_2_O_RB_PLT11_진입OK AT %MW94042.10 : BOOL; (* R363_2_O_RB_PLT11_진입OK *)
    R363_2_O_RB_PLT12_진입OK AT %MW94042.11 : BOOL; (* R363_2_O_RB_PLT12_진입OK *)
    R363_2_O_RB_PLT1_진입OK AT %MW94042.0 : BOOL; (* R363_2_O_RB_PLT1_진입OK *)
    R363_2_O_RB_PLT2_진입OK AT %MW94042.1 : BOOL; (* R363_2_O_RB_PLT2_진입OK *)
    R363_2_O_RB_PLT3_진입OK AT %MW94042.2 : BOOL; (* R363_2_O_RB_PLT3_진입OK *)
    R363_2_O_RB_PLT4_진입OK AT %MW94042.3 : BOOL; (* R363_2_O_RB_PLT4_진입OK *)
    R363_2_O_RB_PLT5_진입OK AT %MW94042.4 : BOOL; (* R363_2_O_RB_PLT5_진입OK *)
    R363_2_O_RB_PLT6_진입OK AT %MW94042.5 : BOOL; (* R363_2_O_RB_PLT6_진입OK *)
    R363_2_O_RB_PLT7_진입OK AT %MW94042.6 : BOOL; (* R363_2_O_RB_PLT7_진입OK *)
    R363_2_O_RB_PLT8_진입OK AT %MW94042.7 : BOOL; (* R363_2_O_RB_PLT8_진입OK *)
    R363_2_O_RB_PLT9_진입OK AT %MW94042.8 : BOOL; (* R363_2_O_RB_PLT9_진입OK *)
    R363_2_O_RB_PLT_카운터_리셋_요구 AT %MW94043.10 : BOOL; (* R363_2_O_RB_PLT_카운터_리셋_요구 *)
    R363_2_O_RB_PROG_선택1 AT %MW94040.0 : BOOL; (* R363_2_O_RB_PROG_선택1 *)
    R363_2_O_RB_PROG_선택128 AT %MW94040.7 : BOOL; (* R363_2_O_RB_PROG_선택128 *)
    R363_2_O_RB_PROG_선택16 AT %MW94040.4 : BOOL; (* R363_2_O_RB_PROG_선택16 *)
    R363_2_O_RB_PROG_선택2 AT %MW94040.1 : BOOL; (* R363_2_O_RB_PROG_선택2 *)
    R363_2_O_RB_PROG_선택32 AT %MW94040.5 : BOOL; (* R363_2_O_RB_PROG_선택32 *)
    R363_2_O_RB_PROG_선택4 AT %MW94040.2 : BOOL; (* R363_2_O_RB_PROG_선택4 *)
    R363_2_O_RB_PROG_선택64 AT %MW94040.6 : BOOL; (* R363_2_O_RB_PROG_선택64 *)
    R363_2_O_RB_PROG_선택8 AT %MW94040.3 : BOOL; (* R363_2_O_RB_PROG_선택8 *)
    R363_2_O_RB_SP_1_14 AT %MW94041.14 : BOOL; (* R363_2_O_RB_SP_1_14 *)
    R363_2_O_RB_SP_1_15 AT %MW94041.15 : BOOL; (* R363_2_O_RB_SP_1_15 *)
    R363_2_O_RB_SP_2_12 AT %MW94042.12 : BOOL; (* R363_2_O_RB_SP_2_12 *)
    R363_2_O_RB_SP_2_13 AT %MW94042.13 : BOOL; (* R363_2_O_RB_SP_2_13 *)
    R363_2_O_RB_SP_2_14 AT %MW94042.14 : BOOL; (* R363_2_O_RB_SP_2_14 *)
    R363_2_O_RB_SP_5000TH_ON AT %MW94042.15 : BOOL; (* R363_2_O_RB_SP_5000TH_ON *)
    R363_2_O_RB_TIP_CHANGE_END AT %MW94043.9 : BOOL; (* R363_2_O_RB_TIP_CHANGE_END *)
    R363_2_O_RB_TIP_CHANGE_START AT %MW94043.8 : BOOL; (* R363_2_O_RB_TIP_CHANGE_START *)
    R363_2_O_RB_TIP_DRESS_SATRT AT %MW94040.12 : BOOL; (* R363_2_O_RB_TIP_DRESS_SATRT *)
    R363_2_O_RB_VIP_MODE AT %MW94043.15 : BOOL; (* R363_2_O_RB_VIP_MODE *)
    R363_2_O_RB_기동 AT %MW94040.9 : BOOL; (* R363_2_O_RB_기동 *)
    R363_2_O_RB_냉각수차단 AT %MW94040.15 : BOOL; (* R363_2_O_RB_냉각수차단 *)
    R363_2_O_RB_부저정지 AT %MW94043.13 : BOOL; (* R363_2_O_RB_부저정지 *)
    R363_2_O_RB_비상정지_NC AT %MW94043.12 : BOOL; (* R363_2_O_RB_비상정지_NC *)
    R363_2_O_RB_상호인터록_INT1 AT %MW94043.0 : BOOL; (* R363_2_O_RB_상호인터록_INT1 *)
    R363_2_O_RB_상호인터록_INT2 AT %MW94043.1 : BOOL; (* R363_2_O_RB_상호인터록_INT2 *)
    R363_2_O_RB_상호인터록_INT3 AT %MW94043.2 : BOOL; (* R363_2_O_RB_상호인터록_INT3 *)
    R363_2_O_RB_상호인터록_INT4 AT %MW94043.3 : BOOL; (* R363_2_O_RB_상호인터록_INT4 *)
    R363_2_O_RB_상호인터록_INT5 AT %MW94043.4 : BOOL; (* R363_2_O_RB_상호인터록_INT5 *)
    R363_2_O_RB_상호인터록_INT6 AT %MW94043.5 : BOOL; (* R363_2_O_RB_상호인터록_INT6 *)
    R363_2_O_RB_상호인터록_INT7 AT %MW94043.6 : BOOL; (* R363_2_O_RB_상호인터록_INT7 *)
    R363_2_O_RB_상호인터록_INT8 AT %MW94043.7 : BOOL; (* R363_2_O_RB_상호인터록_INT8 *)
    R363_2_O_RB_이상_리셋 AT %MW94040.10 : BOOL; (* R363_2_O_RB_이상_리셋 *)
    R363_2_O_RB_작업완료_리셋 AT %MW94040.8 : BOOL; (* R363_2_O_RB_작업완료_리셋 *)
    R364_1_I_RB_0_5_COMM_CHK AT %MW84053.14 : BOOL; (* R364_1_I_RB_0_5_COMM_CHK *)
    R364_1_I_RB_10차_간섭무 AT %MW84051.9 : BOOL; (* R364_1_I_RB_10차_간섭무 *)
    R364_1_I_RB_11차_간섭무 AT %MW84051.10 : BOOL; (* R364_1_I_RB_11차_간섭무 *)
    R364_1_I_RB_12차_간섭무 AT %MW84051.11 : BOOL; (* R364_1_I_RB_12차_간섭무 *)
    R364_1_I_RB_1차_간섭무 AT %MW84051.0 : BOOL; (* R364_1_I_RB_1차_간섭무 *)
    R364_1_I_RB_1차_작업완료 AT %MW84050.9 : BOOL; (* R364_1_I_RB_1차_작업완료 *)
    R364_1_I_RB_2차_간섭무 AT %MW84051.1 : BOOL; (* R364_1_I_RB_2차_간섭무 *)
    R364_1_I_RB_2차_작업완료 AT %MW84050.10 : BOOL; (* R364_1_I_RB_2차_작업완료 *)
    R364_1_I_RB_3차_간섭무 AT %MW84051.2 : BOOL; (* R364_1_I_RB_3차_간섭무 *)
    R364_1_I_RB_3차_작업완료 AT %MW84050.11 : BOOL; (* R364_1_I_RB_3차_작업완료 *)
    R364_1_I_RB_4차_간섭무 AT %MW84051.3 : BOOL; (* R364_1_I_RB_4차_간섭무 *)
    R364_1_I_RB_4차_작업완료 AT %MW84050.12 : BOOL; (* R364_1_I_RB_4차_작업완료 *)
    R364_1_I_RB_5차_간섭무 AT %MW84051.4 : BOOL; (* R364_1_I_RB_5차_간섭무 *)
    R364_1_I_RB_5차_작업완료 AT %MW84050.13 : BOOL; (* R364_1_I_RB_5차_작업완료 *)
    R364_1_I_RB_6차_간섭무 AT %MW84051.5 : BOOL; (* R364_1_I_RB_6차_간섭무 *)
    R364_1_I_RB_6차_작업완료 AT %MW84050.14 : BOOL; (* R364_1_I_RB_6차_작업완료 *)
    R364_1_I_RB_7차_간섭무 AT %MW84051.6 : BOOL; (* R364_1_I_RB_7차_간섭무 *)
    R364_1_I_RB_7차_작업완료 AT %MW84050.15 : BOOL; (* R364_1_I_RB_7차_작업완료 *)
    R364_1_I_RB_8차_간섭무 AT %MW84051.7 : BOOL; (* R364_1_I_RB_8차_간섭무 *)
    R364_1_I_RB_9차_간섭무 AT %MW84051.8 : BOOL; (* R364_1_I_RB_9차_간섭무 *)
    R364_1_I_RB_AB_NORMAL_선택 AT %MW84050.6 : BOOL; (* R364_1_I_RB_AB_NORMAL_선택 *)
    R364_1_I_RB_GUN1_FIXED_TIP AT %MW84057 : WORD; (* R364_1_I_RB_GUN1_FIXED_TIP *)
    R364_1_I_RB_GUN1_MOVING_TIP AT %MW84056 : WORD; (* R364_1_I_RB_GUN1_MOVING_TIP *)
    R364_1_I_RB_GUN2_FIXED_TIP AT %MW84059 : WORD; (* R364_1_I_RB_GUN2_FIXED_TIP *)
    R364_1_I_RB_GUN2_MOVING_TIP AT %MW84058 : WORD; (* R364_1_I_RB_GUN2_MOVING_TIP *)
    R364_1_I_RB_INPUT AT %MW84050 : ARRAY[0..3] OF WORD; (* R364_1_I_RB_INPUT *)
    R364_1_I_RB_LS_이상 AT %MW84052.11 : BOOL; (* R364_1_I_RB_LS_이상 *)
    R364_1_I_RB_MOTOR_MC_ON AT %MW84053.15 : BOOL; (* R364_1_I_RB_MOTOR_MC_ON *)
    R364_1_I_RB_PLT_UNLOAD_완료 AT %MW84053.11 : BOOL; (* R364_1_I_RB_PLT_UNLOAD_완료 *)
    R364_1_I_RB_PLT_최종UNLOAD_완료 AT %MW84053.12 : BOOL; (* R364_1_I_RB_PLT_최종UNLOAD_완료 *)
    R364_1_I_RB_PROG_ECHO_1 AT %MW84052.0 : BOOL; (* R364_1_I_RB_PROG_ECHO_1 *)
    R364_1_I_RB_PROG_ECHO_128 AT %MW84052.7 : BOOL; (* R364_1_I_RB_PROG_ECHO_128 *)
    R364_1_I_RB_PROG_ECHO_16 AT %MW84052.4 : BOOL; (* R364_1_I_RB_PROG_ECHO_16 *)
    R364_1_I_RB_PROG_ECHO_2 AT %MW84052.1 : BOOL; (* R364_1_I_RB_PROG_ECHO_2 *)
    R364_1_I_RB_PROG_ECHO_32 AT %MW84052.5 : BOOL; (* R364_1_I_RB_PROG_ECHO_32 *)
    R364_1_I_RB_PROG_ECHO_4 AT %MW84052.2 : BOOL; (* R364_1_I_RB_PROG_ECHO_4 *)
    R364_1_I_RB_PROG_ECHO_64 AT %MW84052.6 : BOOL; (* R364_1_I_RB_PROG_ECHO_64 *)
    R364_1_I_RB_PROG_ECHO_8 AT %MW84052.3 : BOOL; (* R364_1_I_RB_PROG_ECHO_8 *)
    R364_1_I_RB_SP3_8 AT %MW84053.8 : BOOL; (* R364_1_I_RB_SP3_8 *)
    R364_1_I_RB_SP3_9 AT %MW84053.9 : BOOL; (* R364_1_I_RB_SP3_9 *)
    R364_1_I_RB_SPARE_WORD_4 AT %MW84054 : WORD; (* R364_1_I_RB_SPARE_WORD_4 *)
    R364_1_I_RB_SP_1_12 AT %MW84051.12 : BOOL; (* R364_1_I_RB_SP_1_12 *)
    R364_1_I_RB_SP_1_13 AT %MW84051.13 : BOOL; (* R364_1_I_RB_SP_1_13 *)
    R364_1_I_RB_SP_1_14 AT %MW84051.14 : BOOL; (* R364_1_I_RB_SP_1_14 *)
    R364_1_I_RB_SP_1_15 AT %MW84051.15 : BOOL; (* R364_1_I_RB_SP_1_15 *)
    R364_1_I_RB_TC_이상 AT %MW84052.8 : BOOL; (* R364_1_I_RB_TC_이상 *)
    R364_1_I_RB_TIP_CHANGE AT %MW84053.13 : BOOL; (* R364_1_I_RB_TIP_CHANGE *)
    R364_1_I_RB_TIP_DRESSING AT %MW84050.7 : BOOL; (* R364_1_I_RB_TIP_DRESSING *)
    R364_1_I_RB__PLT_카운터리셋완료 AT %MW84053.10 : BOOL; (* R364_1_I_RB__PLT_카운터리셋완료 *)
    R364_1_I_RB_공기압_이상 AT %MW84052.9 : BOOL; (* R364_1_I_RB_공기압_이상 *)
    R364_1_I_RB_냉각수_이상 AT %MW84052.10 : BOOL; (* R364_1_I_RB_냉각수_이상 *)
    R364_1_I_RB_비상정지_NC AT %MW84050.8 : BOOL; (* R364_1_I_RB_비상정지_NC *)
    R364_1_I_RB_비전이상 AT %MW84052.14 : BOOL; (* R364_1_I_RB_비전이상 *)
    R364_1_I_RB_상호인터록_INT1 AT %MW84053.0 : BOOL; (* R364_1_I_RB_상호인터록_INT1 *)
    R364_1_I_RB_상호인터록_INT2 AT %MW84053.1 : BOOL; (* R364_1_I_RB_상호인터록_INT2 *)
    R364_1_I_RB_상호인터록_INT3 AT %MW84053.2 : BOOL; (* R364_1_I_RB_상호인터록_INT3 *)
    R364_1_I_RB_상호인터록_INT4 AT %MW84053.3 : BOOL; (* R364_1_I_RB_상호인터록_INT4 *)
    R364_1_I_RB_상호인터록_INT5 AT %MW84053.4 : BOOL; (* R364_1_I_RB_상호인터록_INT5 *)
    R364_1_I_RB_상호인터록_INT6 AT %MW84053.5 : BOOL; (* R364_1_I_RB_상호인터록_INT6 *)
    R364_1_I_RB_상호인터록_INT7 AT %MW84053.6 : BOOL; (* R364_1_I_RB_상호인터록_INT7 *)
    R364_1_I_RB_상호인터록_INT8 AT %MW84053.7 : BOOL; (* R364_1_I_RB_상호인터록_INT8 *)
    R364_1_I_RB_실러이상 AT %MW84052.13 : BOOL; (* R364_1_I_RB_실러이상 *)
    R364_1_I_RB_용접카운터이상 AT %MW84052.15 : BOOL; (* R364_1_I_RB_용접카운터이상 *)
    R364_1_I_RB_용접타점수 AT %MW84055 : WORD; (* R364_1_I_RB_용접타점수 *)
    R364_1_I_RB_운전준비 AT %MW84050.3 : BOOL; (* R364_1_I_RB_운전준비 *)
    R364_1_I_RB_원위치 AT %MW84050.0 : BOOL; (* R364_1_I_RB_원위치 *)
    R364_1_I_RB_이상리셋 AT %MW84050.2 : BOOL; (* R364_1_I_RB_이상리셋 *)
    R364_1_I_RB_자동 AT %MW84050.4 : BOOL; (* R364_1_I_RB_자동 *)
    R364_1_I_RB_자동기동 AT %MW84050.5 : BOOL; (* R364_1_I_RB_자동기동 *)
    R364_1_I_RB_최종_작업완료 AT %MW84050.1 : BOOL; (* R364_1_I_RB_최종_작업완료 *)
    R364_1_I_RB_통신이상 AT %MW84052.12 : BOOL; (* R364_1_I_RB_통신이상 *)
    R364_1_M_I_RB_1차_작업완료 AT %MW20051.2 : BOOL; (* R364_1_M_I_RB_1차_작업완료 *)
    R364_1_M_I_RB_2차_작업완료 AT %MW20051.3 : BOOL; (* R364_1_M_I_RB_2차_작업완료 *)
    R364_1_M_I_RB_3차_작업완료 AT %MW20051.4 : BOOL; (* R364_1_M_I_RB_3차_작업완료 *)
    R364_1_M_I_RB_4차_작업완료 AT %MW20051.5 : BOOL; (* R364_1_M_I_RB_4차_작업완료 *)
    R364_1_M_I_RB_5차_작업완료 AT %MW20051.6 : BOOL; (* R364_1_M_I_RB_5차_작업완료 *)
    R364_1_M_I_RB_6차_작업완료 AT %MW20051.7 : BOOL; (* R364_1_M_I_RB_6차_작업완료 *)
    R364_1_M_I_RB_7차_작업완료 AT %MW20051.8 : BOOL; (* R364_1_M_I_RB_7차_작업완료 *)
    R364_1_M_I_RB_PAUSE_보조 AT %MW20050.5 : BOOL; (* R364_1_M_I_RB_PAUSE_보조 *)
    R364_1_M_I_RB_PLC_RUN_CHK_이상 AT %MW20050.7 : BOOL; (* R364_1_M_I_RB_PLC_RUN_CHK_이상 *)
    R364_1_M_I_RB_간섭무_1 AT %MW20052.0 : BOOL; (* R364_1_M_I_RB_간섭무_1 *)
    R364_1_M_I_RB_간섭무_10 AT %MW20052.9 : BOOL; (* R364_1_M_I_RB_간섭무_10 *)
    R364_1_M_I_RB_간섭무_11 AT %MW20052.10 : BOOL; (* R364_1_M_I_RB_간섭무_11 *)
    R364_1_M_I_RB_간섭무_12 AT %MW20052.11 : BOOL; (* R364_1_M_I_RB_간섭무_12 *)
    R364_1_M_I_RB_간섭무_2 AT %MW20052.1 : BOOL; (* R364_1_M_I_RB_간섭무_2 *)
    R364_1_M_I_RB_간섭무_3 AT %MW20052.2 : BOOL; (* R364_1_M_I_RB_간섭무_3 *)
    R364_1_M_I_RB_간섭무_4 AT %MW20052.3 : BOOL; (* R364_1_M_I_RB_간섭무_4 *)
    R364_1_M_I_RB_간섭무_5 AT %MW20052.4 : BOOL; (* R364_1_M_I_RB_간섭무_5 *)
    R364_1_M_I_RB_간섭무_6 AT %MW20052.5 : BOOL; (* R364_1_M_I_RB_간섭무_6 *)
    R364_1_M_I_RB_간섭무_7 AT %MW20052.6 : BOOL; (* R364_1_M_I_RB_간섭무_7 *)
    R364_1_M_I_RB_간섭무_8 AT %MW20052.7 : BOOL; (* R364_1_M_I_RB_간섭무_8 *)
    R364_1_M_I_RB_간섭무_9 AT %MW20052.8 : BOOL; (* R364_1_M_I_RB_간섭무_9 *)
    R364_1_M_I_RB_비상정지 AT %MW20050.4 : BOOL; (* R364_1_M_I_RB_비상정지 *)
    R364_1_M_I_RB_운전준비 AT %MW20050.0 : BOOL; (* R364_1_M_I_RB_운전준비 *)
    R364_1_M_I_RB_원위치 AT %MW20050.3 : BOOL; (* R364_1_M_I_RB_원위치 *)
    R364_1_M_I_RB_이상 AT %MW20050.2 : BOOL; (* R364_1_M_I_RB_이상 *)
    R364_1_M_I_RB_자동 AT %MW20050.1 : BOOL; (* R364_1_M_I_RB_자동 *)
    R364_1_M_I_RB_최종작업완료 AT %MW20051.0 : BOOL; (* R364_1_M_I_RB_최종작업완료 *)
    R364_1_M_I_RB_프로그램_이상 AT %MW20050.6 : BOOL; (* R364_1_M_I_RB_프로그램_이상 *)
    R364_1_M_O_RB_1_CYCLE_SET AT %MW21050.3 : BOOL; (* R364_1_M_O_RB_1_CYCLE_SET *)
    R364_1_M_O_RB_1_CYCLE_리셋 AT %MW21050.4 : BOOL; (* R364_1_M_O_RB_1_CYCLE_리셋 *)
    R364_1_M_O_RB_1차_작업완료_리셋 AT %MW21052.0 : BOOL; (* R364_1_M_O_RB_1차_작업완료_리셋 *)
    R364_1_M_O_RB_2차_작업완료_리셋 AT %MW21052.1 : BOOL; (* R364_1_M_O_RB_2차_작업완료_리셋 *)
    R364_1_M_O_RB_2차_진입OK AT %MW21051.8 : BOOL; (* R364_1_M_O_RB_2차_진입OK *)
    R364_1_M_O_RB_3차_작업완료_리셋 AT %MW21052.2 : BOOL; (* R364_1_M_O_RB_3차_작업완료_리셋 *)
    R364_1_M_O_RB_3차_진입OK AT %MW21051.9 : BOOL; (* R364_1_M_O_RB_3차_진입OK *)
    R364_1_M_O_RB_4차_작업완료_리셋 AT %MW21052.3 : BOOL; (* R364_1_M_O_RB_4차_작업완료_리셋 *)
    R364_1_M_O_RB_4차_진입OK AT %MW21051.10 : BOOL; (* R364_1_M_O_RB_4차_진입OK *)
    R364_1_M_O_RB_5차_작업완료_리셋 AT %MW21052.4 : BOOL; (* R364_1_M_O_RB_5차_작업완료_리셋 *)
    R364_1_M_O_RB_5차_진입OK AT %MW21051.11 : BOOL; (* R364_1_M_O_RB_5차_진입OK *)
    R364_1_M_O_RB_6차_작업완료_리셋 AT %MW21052.5 : BOOL; (* R364_1_M_O_RB_6차_작업완료_리셋 *)
    R364_1_M_O_RB_6차_진입OK AT %MW21051.12 : BOOL; (* R364_1_M_O_RB_6차_진입OK *)
    R364_1_M_O_RB_7차_작업완료_리셋 AT %MW21052.6 : BOOL; (* R364_1_M_O_RB_7차_작업완료_리셋 *)
    R364_1_M_O_RB_7차_진입OK AT %MW21051.13 : BOOL; (* R364_1_M_O_RB_7차_진입OK *)
    R364_1_M_O_RB_ATD_OK AT %MW21050.6 : BOOL; (* R364_1_M_O_RB_ATD_OK *)
    R364_1_M_O_RB_PLT_10_진입OK AT %MW21053.10 : BOOL; (* R364_1_M_O_RB_PLT_10_진입OK *)
    R364_1_M_O_RB_PLT_11_진입OK AT %MW21053.11 : BOOL; (* R364_1_M_O_RB_PLT_11_진입OK *)
    R364_1_M_O_RB_PLT_12_진입OK AT %MW21053.12 : BOOL; (* R364_1_M_O_RB_PLT_12_진입OK *)
    R364_1_M_O_RB_PLT_1_진입OK AT %MW21053.1 : BOOL; (* R364_1_M_O_RB_PLT_1_진입OK *)
    R364_1_M_O_RB_PLT_2_진입OK AT %MW21053.2 : BOOL; (* R364_1_M_O_RB_PLT_2_진입OK *)
    R364_1_M_O_RB_PLT_3_진입OK AT %MW21053.3 : BOOL; (* R364_1_M_O_RB_PLT_3_진입OK *)
    R364_1_M_O_RB_PLT_4_진입OK AT %MW21053.4 : BOOL; (* R364_1_M_O_RB_PLT_4_진입OK *)
    R364_1_M_O_RB_PLT_5_진입OK AT %MW21053.5 : BOOL; (* R364_1_M_O_RB_PLT_5_진입OK *)
    R364_1_M_O_RB_PLT_6_진입OK AT %MW21053.6 : BOOL; (* R364_1_M_O_RB_PLT_6_진입OK *)
    R364_1_M_O_RB_PLT_7_진입OK AT %MW21053.7 : BOOL; (* R364_1_M_O_RB_PLT_7_진입OK *)
    R364_1_M_O_RB_PLT_8_진입OK AT %MW21053.8 : BOOL; (* R364_1_M_O_RB_PLT_8_진입OK *)
    R364_1_M_O_RB_PLT_9_진입OK AT %MW21053.9 : BOOL; (* R364_1_M_O_RB_PLT_9_진입OK *)
    R364_1_M_O_RB_PLT_카운터리셋_보조 AT %MW21050.10 : BOOL; (* R364_1_M_O_RB_PLT_카운터리셋_보조 *)
    R364_1_M_O_RB_PROG_NO AT %MW21054 : WORD;
    R364_1_M_O_RB_RESTART_OK AT %MW21050.2 : BOOL; (* R364_1_M_O_RB_RESTART_OK *)
    R364_1_M_O_RB_START_OK AT %MW21050.0 : BOOL; (* R364_1_M_O_RB_START_OK *)
    R364_1_M_O_RB_TEST_MODE_5000회 AT %MW21050.12 : BOOL; (* R364_1_M_O_RB_TEST_MODE_5000회 *)
    R364_1_M_O_RB_TIP_교체_시작 AT %MW21050.7 : BOOL; (* R364_1_M_O_RB_TIP_교체_시작 *)
    R364_1_M_O_RB_TIP_교체_완료 AT %MW21050.8 : BOOL; (* R364_1_M_O_RB_TIP_교체_완료 *)
    R364_1_M_O_RB_VIP_MODE AT %MW21050.11 : BOOL; (* R364_1_M_O_RB_VIP_MODE *)
    R364_1_M_O_RB_냉각수_차단_요청 AT %MW21050.9 : BOOL; (* R364_1_M_O_RB_냉각수_차단_요청 *)
    R364_1_M_O_RB_진입OK_AX차종 AT %MW21051.0 : BOOL; (* R364_1_M_O_RB_진입OK_AX차종 *)
    R364_1_M_O_RB_진입OK_B차종 AT %MW21051.1 : BOOL; (* R364_1_M_O_RB_진입OK_B차종 *)
    R364_1_M_O_RB_진입OK_C차종 AT %MW21051.2 : BOOL; (* R364_1_M_O_RB_진입OK_C차종 *)
    R364_1_M_O_RB_진입OK_D차종 AT %MW21051.3 : BOOL; (* R364_1_M_O_RB_진입OK_D차종 *)
    R364_1_M_O_RB_진입OK_E차종 AT %MW21051.4 : BOOL; (* R364_1_M_O_RB_진입OK_E차종 *)
    R364_1_M_O_RB_진입OK_F차종 AT %MW21051.5 : BOOL; (* R364_1_M_O_RB_진입OK_F차종 *)
    R364_1_M_O_RB_진입OK_G차종 AT %MW21051.6 : BOOL; (* R364_1_M_O_RB_진입OK_G차종 *)
    R364_1_M_O_RB_진입OK_H차종 AT %MW21051.7 : BOOL; (* R364_1_M_O_RB_진입OK_H차종 *)
    R364_1_M_O_RB_최종_작업완료_리셋 AT %MW21050.5 : BOOL; (* R364_1_M_O_RB_최종_작업완료_리셋 *)
    R364_1_M_O_RB_프로그램_OK AT %MW21050.1 : BOOL; (* R364_1_M_O_RB_프로그램_OK *)
    R364_1_O_RB_0_5S_통신_CHK AT %MW94053.14 : BOOL; (* R364_1_O_RB_0_5S_통신_CHK *)
    R364_1_O_RB_2차_진입OK AT %MW94051.8 : BOOL; (* R364_1_O_RB_2차_진입OK *)
    R364_1_O_RB_3차_진입OK AT %MW94051.9 : BOOL; (* R364_1_O_RB_3차_진입OK *)
    R364_1_O_RB_4차_진입OK AT %MW94051.10 : BOOL; (* R364_1_O_RB_4차_진입OK *)
    R364_1_O_RB_5차_진입OK AT %MW94051.11 : BOOL; (* R364_1_O_RB_5차_진입OK *)
    R364_1_O_RB_6차_진입OK AT %MW94051.12 : BOOL; (* R364_1_O_RB_6차_진입OK *)
    R364_1_O_RB_7차_진입OK AT %MW94051.13 : BOOL; (* R364_1_O_RB_7차_진입OK *)
    R364_1_O_RB_AX_1차_진입OK AT %MW94051.0 : BOOL; (* R364_1_O_RB_AX_1차_진입OK *)
    R364_1_O_RB_B_1차_진입OK AT %MW94051.1 : BOOL; (* R364_1_O_RB_B_1차_진입OK *)
    R364_1_O_RB_C_1차_진입OK AT %MW94051.2 : BOOL; (* R364_1_O_RB_C_1차_진입OK *)
    R364_1_O_RB_D_1차_진입OK AT %MW94051.3 : BOOL; (* R364_1_O_RB_D_1차_진입OK *)
    R364_1_O_RB_EACH_작업완료_리셋 AT %MW94050.14 : BOOL; (* R364_1_O_RB_EACH_작업완료_리셋 *)
    R364_1_O_RB_EXT_READY AT %MW94050.11 : BOOL; (* R364_1_O_RB_EXT_READY *)
    R364_1_O_RB_E_1차_진입OK AT %MW94051.4 : BOOL; (* R364_1_O_RB_E_1차_진입OK *)
    R364_1_O_RB_F_1차_진입OK AT %MW94051.5 : BOOL; (* R364_1_O_RB_F_1차_진입OK *)
    R364_1_O_RB_GATE_OPEN_NC AT %MW94053.11 : BOOL; (* R364_1_O_RB_GATE_OPEN_NC *)
    R364_1_O_RB_G_1차_진입OK AT %MW94051.6 : BOOL; (* R364_1_O_RB_G_1차_진입OK *)
    R364_1_O_RB_H_1차_진입OK AT %MW94051.7 : BOOL; (* R364_1_O_RB_H_1차_진입OK *)
    R364_1_O_RB_OUTPUT AT %MW94050 : ARRAY[0..3] OF WORD; (* R364_1_O_RB_OUTPUT *)
    R364_1_O_RB_PAUSE_NC AT %MW94050.13 : BOOL; (* R364_1_O_RB_PAUSE_NC *)
    R364_1_O_RB_PLT10_진입OK AT %MW94052.9 : BOOL; (* R364_1_O_RB_PLT10_진입OK *)
    R364_1_O_RB_PLT11_진입OK AT %MW94052.10 : BOOL; (* R364_1_O_RB_PLT11_진입OK *)
    R364_1_O_RB_PLT12_진입OK AT %MW94052.11 : BOOL; (* R364_1_O_RB_PLT12_진입OK *)
    R364_1_O_RB_PLT1_진입OK AT %MW94052.0 : BOOL; (* R364_1_O_RB_PLT1_진입OK *)
    R364_1_O_RB_PLT2_진입OK AT %MW94052.1 : BOOL; (* R364_1_O_RB_PLT2_진입OK *)
    R364_1_O_RB_PLT3_진입OK AT %MW94052.2 : BOOL; (* R364_1_O_RB_PLT3_진입OK *)
    R364_1_O_RB_PLT4_진입OK AT %MW94052.3 : BOOL; (* R364_1_O_RB_PLT4_진입OK *)
    R364_1_O_RB_PLT5_진입OK AT %MW94052.4 : BOOL; (* R364_1_O_RB_PLT5_진입OK *)
    R364_1_O_RB_PLT6_진입OK AT %MW94052.5 : BOOL; (* R364_1_O_RB_PLT6_진입OK *)
    R364_1_O_RB_PLT7_진입OK AT %MW94052.6 : BOOL; (* R364_1_O_RB_PLT7_진입OK *)
    R364_1_O_RB_PLT8_진입OK AT %MW94052.7 : BOOL; (* R364_1_O_RB_PLT8_진입OK *)
    R364_1_O_RB_PLT9_진입OK AT %MW94052.8 : BOOL; (* R364_1_O_RB_PLT9_진입OK *)
    R364_1_O_RB_PLT_카운터_리셋_요구 AT %MW94053.10 : BOOL; (* R364_1_O_RB_PLT_카운터_리셋_요구 *)
    R364_1_O_RB_PROG_선택1 AT %MW94050.0 : BOOL; (* R364_1_O_RB_PROG_선택1 *)
    R364_1_O_RB_PROG_선택128 AT %MW94050.7 : BOOL; (* R364_1_O_RB_PROG_선택128 *)
    R364_1_O_RB_PROG_선택16 AT %MW94050.4 : BOOL; (* R364_1_O_RB_PROG_선택16 *)
    R364_1_O_RB_PROG_선택2 AT %MW94050.1 : BOOL; (* R364_1_O_RB_PROG_선택2 *)
    R364_1_O_RB_PROG_선택32 AT %MW94050.5 : BOOL; (* R364_1_O_RB_PROG_선택32 *)
    R364_1_O_RB_PROG_선택4 AT %MW94050.2 : BOOL; (* R364_1_O_RB_PROG_선택4 *)
    R364_1_O_RB_PROG_선택64 AT %MW94050.6 : BOOL; (* R364_1_O_RB_PROG_선택64 *)
    R364_1_O_RB_PROG_선택8 AT %MW94050.3 : BOOL; (* R364_1_O_RB_PROG_선택8 *)
    R364_1_O_RB_SP_1_14 AT %MW94051.14 : BOOL; (* R364_1_O_RB_SP_1_14 *)
    R364_1_O_RB_SP_1_15 AT %MW94051.15 : BOOL; (* R364_1_O_RB_SP_1_15 *)
    R364_1_O_RB_SP_2_12 AT %MW94052.12 : BOOL; (* R364_1_O_RB_SP_2_12 *)
    R364_1_O_RB_SP_2_13 AT %MW94052.13 : BOOL; (* R364_1_O_RB_SP_2_13 *)
    R364_1_O_RB_SP_2_14 AT %MW94052.14 : BOOL; (* R364_1_O_RB_SP_2_14 *)
    R364_1_O_RB_SP_5000TH_ON AT %MW94052.15 : BOOL; (* R364_1_O_RB_SP_5000TH_ON *)
    R364_1_O_RB_TIP_CHANGE_END AT %MW94053.9 : BOOL; (* R364_1_O_RB_TIP_CHANGE_END *)
    R364_1_O_RB_TIP_CHANGE_START AT %MW94053.8 : BOOL; (* R364_1_O_RB_TIP_CHANGE_START *)
    R364_1_O_RB_TIP_DRESS_SATRT AT %MW94050.12 : BOOL; (* R364_1_O_RB_TIP_DRESS_SATRT *)
    R364_1_O_RB_VIP_MODE AT %MW94053.15 : BOOL; (* R364_1_O_RB_VIP_MODE *)
    R364_1_O_RB_기동 AT %MW94050.9 : BOOL; (* R364_1_O_RB_기동 *)
    R364_1_O_RB_냉각수차단 AT %MW94050.15 : BOOL; (* R364_1_O_RB_냉각수차단 *)
    R364_1_O_RB_부저정지 AT %MW94053.13 : BOOL; (* R364_1_O_RB_부저정지 *)
    R364_1_O_RB_비상정지_NC AT %MW94053.12 : BOOL; (* R364_1_O_RB_비상정지_NC *)
    R364_1_O_RB_상호인터록_INT1 AT %MW94053.0 : BOOL; (* R364_1_O_RB_상호인터록_INT1 *)
    R364_1_O_RB_상호인터록_INT2 AT %MW94053.1 : BOOL; (* R364_1_O_RB_상호인터록_INT2 *)
    R364_1_O_RB_상호인터록_INT3 AT %MW94053.2 : BOOL; (* R364_1_O_RB_상호인터록_INT3 *)
    R364_1_O_RB_상호인터록_INT4 AT %MW94053.3 : BOOL; (* R364_1_O_RB_상호인터록_INT4 *)
    R364_1_O_RB_상호인터록_INT5 AT %MW94053.4 : BOOL; (* R364_1_O_RB_상호인터록_INT5 *)
    R364_1_O_RB_상호인터록_INT6 AT %MW94053.5 : BOOL; (* R364_1_O_RB_상호인터록_INT6 *)
    R364_1_O_RB_상호인터록_INT7 AT %MW94053.6 : BOOL; (* R364_1_O_RB_상호인터록_INT7 *)
    R364_1_O_RB_상호인터록_INT8 AT %MW94053.7 : BOOL; (* R364_1_O_RB_상호인터록_INT8 *)
    R364_1_O_RB_이상_리셋 AT %MW94050.10 : BOOL; (* R364_1_O_RB_이상_리셋 *)
    R364_1_O_RB_작업완료_리셋 AT %MW94050.8 : BOOL; (* R364_1_O_RB_작업완료_리셋 *)
    R366_1_I_RB_0_5_COMM_CHK AT %MW84063.14 : BOOL; (* R366_1_I_RB_0_5_COMM_CHK *)
    R366_1_I_RB_10차_간섭무 AT %MW84061.9 : BOOL; (* R366_1_I_RB_10차_간섭무 *)
    R366_1_I_RB_11차_간섭무 AT %MW84061.10 : BOOL; (* R366_1_I_RB_11차_간섭무 *)
    R366_1_I_RB_12차_간섭무 AT %MW84061.11 : BOOL; (* R366_1_I_RB_12차_간섭무 *)
    R366_1_I_RB_1차_간섭무 AT %MW84061.0 : BOOL; (* R366_1_I_RB_1차_간섭무 *)
    R366_1_I_RB_1차_작업완료 AT %MW84060.9 : BOOL; (* R366_1_I_RB_1차_작업완료 *)
    R366_1_I_RB_2차_간섭무 AT %MW84061.1 : BOOL; (* R366_1_I_RB_2차_간섭무 *)
    R366_1_I_RB_2차_작업완료 AT %MW84060.10 : BOOL; (* R366_1_I_RB_2차_작업완료 *)
    R366_1_I_RB_3차_간섭무 AT %MW84061.2 : BOOL; (* R366_1_I_RB_3차_간섭무 *)
    R366_1_I_RB_3차_작업완료 AT %MW84060.11 : BOOL; (* R366_1_I_RB_3차_작업완료 *)
    R366_1_I_RB_4차_간섭무 AT %MW84061.3 : BOOL; (* R366_1_I_RB_4차_간섭무 *)
    R366_1_I_RB_4차_작업완료 AT %MW84060.12 : BOOL; (* R366_1_I_RB_4차_작업완료 *)
    R366_1_I_RB_5차_간섭무 AT %MW84061.4 : BOOL; (* R366_1_I_RB_5차_간섭무 *)
    R366_1_I_RB_5차_작업완료 AT %MW84060.13 : BOOL; (* R366_1_I_RB_5차_작업완료 *)
    R366_1_I_RB_6차_간섭무 AT %MW84061.5 : BOOL; (* R366_1_I_RB_6차_간섭무 *)
    R366_1_I_RB_6차_작업완료 AT %MW84060.14 : BOOL; (* R366_1_I_RB_6차_작업완료 *)
    R366_1_I_RB_7차_간섭무 AT %MW84061.6 : BOOL; (* R366_1_I_RB_7차_간섭무 *)
    R366_1_I_RB_7차_작업완료 AT %MW84060.15 : BOOL; (* R366_1_I_RB_7차_작업완료 *)
    R366_1_I_RB_8차_간섭무 AT %MW84061.7 : BOOL; (* R366_1_I_RB_8차_간섭무 *)
    R366_1_I_RB_9차_간섭무 AT %MW84061.8 : BOOL; (* R366_1_I_RB_9차_간섭무 *)
    R366_1_I_RB_AB_NORMAL_선택 AT %MW84060.6 : BOOL; (* R366_1_I_RB_AB_NORMAL_선택 *)
    R366_1_I_RB_GUN1_FIXED_TIP AT %MW84067 : WORD; (* R366_1_I_RB_GUN1_FIXED_TIP *)
    R366_1_I_RB_GUN1_MOVING_TIP AT %MW84066 : WORD; (* R366_1_I_RB_GUN1_MOVING_TIP *)
    R366_1_I_RB_GUN2_FIXED_TIP AT %MW84069 : WORD; (* R366_1_I_RB_GUN2_FIXED_TIP *)
    R366_1_I_RB_GUN2_MOVING_TIP AT %MW84068 : WORD; (* R366_1_I_RB_GUN2_MOVING_TIP *)
    R366_1_I_RB_INPUT AT %MW84060 : ARRAY[0..3] OF WORD; (* R366_1_I_RB_INPUT *)
    R366_1_I_RB_LS_이상 AT %MW84062.11 : BOOL; (* R366_1_I_RB_LS_이상 *)
    R366_1_I_RB_MOTOR_MC_ON AT %MW84063.15 : BOOL; (* R366_1_I_RB_MOTOR_MC_ON *)
    R366_1_I_RB_PLT_UNLOAD_완료 AT %MW84063.11 : BOOL; (* R366_1_I_RB_PLT_UNLOAD_완료 *)
    R366_1_I_RB_PLT_최종UNLOAD_완료 AT %MW84063.12 : BOOL; (* R366_1_I_RB_PLT_최종UNLOAD_완료 *)
    R366_1_I_RB_PROG_ECHO_1 AT %MW84062.0 : BOOL; (* R366_1_I_RB_PROG_ECHO_1 *)
    R366_1_I_RB_PROG_ECHO_128 AT %MW84062.7 : BOOL; (* R366_1_I_RB_PROG_ECHO_128 *)
    R366_1_I_RB_PROG_ECHO_16 AT %MW84062.4 : BOOL; (* R366_1_I_RB_PROG_ECHO_16 *)
    R366_1_I_RB_PROG_ECHO_2 AT %MW84062.1 : BOOL; (* R366_1_I_RB_PROG_ECHO_2 *)
    R366_1_I_RB_PROG_ECHO_32 AT %MW84062.5 : BOOL; (* R366_1_I_RB_PROG_ECHO_32 *)
    R366_1_I_RB_PROG_ECHO_4 AT %MW84062.2 : BOOL; (* R366_1_I_RB_PROG_ECHO_4 *)
    R366_1_I_RB_PROG_ECHO_64 AT %MW84062.6 : BOOL; (* R366_1_I_RB_PROG_ECHO_64 *)
    R366_1_I_RB_PROG_ECHO_8 AT %MW84062.3 : BOOL; (* R366_1_I_RB_PROG_ECHO_8 *)
    R366_1_I_RB_SP3_8 AT %MW84063.8 : BOOL; (* R366_1_I_RB_SP3_8 *)
    R366_1_I_RB_SP3_9 AT %MW84063.9 : BOOL; (* R366_1_I_RB_SP3_9 *)
    R366_1_I_RB_SPARE_WORD_4 AT %MW84064 : WORD; (* R366_1_I_RB_SPARE_WORD_4 *)
    R366_1_I_RB_SP_1_12 AT %MW84061.12 : BOOL; (* R366_1_I_RB_SP_1_12 *)
    R366_1_I_RB_SP_1_13 AT %MW84061.13 : BOOL; (* R366_1_I_RB_SP_1_13 *)
    R366_1_I_RB_SP_1_14 AT %MW84061.14 : BOOL; (* R366_1_I_RB_SP_1_14 *)
    R366_1_I_RB_SP_1_15 AT %MW84061.15 : BOOL; (* R366_1_I_RB_SP_1_15 *)
    R366_1_I_RB_TC_이상 AT %MW84062.8 : BOOL; (* R366_1_I_RB_TC_이상 *)
    R366_1_I_RB_TIP_CHANGE AT %MW84063.13 : BOOL; (* R366_1_I_RB_TIP_CHANGE *)
    R366_1_I_RB_TIP_DRESSING AT %MW84060.7 : BOOL; (* R366_1_I_RB_TIP_DRESSING *)
    R366_1_I_RB__PLT_카운터리셋완료 AT %MW84063.10 : BOOL; (* R366_1_I_RB__PLT_카운터리셋완료 *)
    R366_1_I_RB_공기압_이상 AT %MW84062.9 : BOOL; (* R366_1_I_RB_공기압_이상 *)
    R366_1_I_RB_냉각수_이상 AT %MW84062.10 : BOOL; (* R366_1_I_RB_냉각수_이상 *)
    R366_1_I_RB_비상정지_NC AT %MW84060.8 : BOOL; (* R366_1_I_RB_비상정지_NC *)
    R366_1_I_RB_비전이상 AT %MW84062.14 : BOOL; (* R366_1_I_RB_비전이상 *)
    R366_1_I_RB_상호인터록_INT1 AT %MW84063.0 : BOOL; (* R366_1_I_RB_상호인터록_INT1 *)
    R366_1_I_RB_상호인터록_INT2 AT %MW84063.1 : BOOL; (* R366_1_I_RB_상호인터록_INT2 *)
    R366_1_I_RB_상호인터록_INT3 AT %MW84063.2 : BOOL; (* R366_1_I_RB_상호인터록_INT3 *)
    R366_1_I_RB_상호인터록_INT4 AT %MW84063.3 : BOOL; (* R366_1_I_RB_상호인터록_INT4 *)
    R366_1_I_RB_상호인터록_INT5 AT %MW84063.4 : BOOL; (* R366_1_I_RB_상호인터록_INT5 *)
    R366_1_I_RB_상호인터록_INT6 AT %MW84063.5 : BOOL; (* R366_1_I_RB_상호인터록_INT6 *)
    R366_1_I_RB_상호인터록_INT7 AT %MW84063.6 : BOOL; (* R366_1_I_RB_상호인터록_INT7 *)
    R366_1_I_RB_상호인터록_INT8 AT %MW84063.7 : BOOL; (* R366_1_I_RB_상호인터록_INT8 *)
    R366_1_I_RB_실러이상 AT %MW84062.13 : BOOL; (* R366_1_I_RB_실러이상 *)
    R366_1_I_RB_용접카운터이상 AT %MW84062.15 : BOOL; (* R366_1_I_RB_용접카운터이상 *)
    R366_1_I_RB_용접타점수 AT %MW84065 : WORD; (* R366_1_I_RB_용접타점수 *)
    R366_1_I_RB_운전준비 AT %MW84060.3 : BOOL; (* R366_1_I_RB_운전준비 *)
    R366_1_I_RB_원위치 AT %MW84060.0 : BOOL; (* R366_1_I_RB_원위치 *)
    R366_1_I_RB_이상리셋 AT %MW84060.2 : BOOL; (* R366_1_I_RB_이상리셋 *)
    R366_1_I_RB_자동 AT %MW84060.4 : BOOL; (* R366_1_I_RB_자동 *)
    R366_1_I_RB_자동기동 AT %MW84060.5 : BOOL; (* R366_1_I_RB_자동기동 *)
    R366_1_I_RB_최종_작업완료 AT %MW84060.1 : BOOL; (* R366_1_I_RB_최종_작업완료 *)
    R366_1_I_RB_통신이상 AT %MW84062.12 : BOOL; (* R366_1_I_RB_통신이상 *)
    R366_1_M_I_RB_1차_작업완료 AT %MW20061.2 : BOOL; (* R366_1_M_I_RB_1차_작업완료 *)
    R366_1_M_I_RB_2차_작업완료 AT %MW20061.3 : BOOL; (* R366_1_M_I_RB_2차_작업완료 *)
    R366_1_M_I_RB_3차_작업완료 AT %MW20061.4 : BOOL; (* R366_1_M_I_RB_3차_작업완료 *)
    R366_1_M_I_RB_4차_작업완료 AT %MW20061.5 : BOOL; (* R366_1_M_I_RB_4차_작업완료 *)
    R366_1_M_I_RB_5차_작업완료 AT %MW20061.6 : BOOL; (* R366_1_M_I_RB_5차_작업완료 *)
    R366_1_M_I_RB_6차_작업완료 AT %MW20061.7 : BOOL; (* R366_1_M_I_RB_6차_작업완료 *)
    R366_1_M_I_RB_7차_작업완료 AT %MW20061.8 : BOOL; (* R366_1_M_I_RB_7차_작업완료 *)
    R366_1_M_I_RB_PAUSE_보조 AT %MW20060.5 : BOOL; (* R366_1_M_I_RB_PAUSE_보조 *)
    R366_1_M_I_RB_PLC_RUN_CHK_이상 AT %MW20060.7 : BOOL; (* R366_1_M_I_RB_PLC_RUN_CHK_이상 *)
    R366_1_M_I_RB_간섭무_1 AT %MW20062.0 : BOOL; (* R366_1_M_I_RB_간섭무_1 *)
    R366_1_M_I_RB_간섭무_10 AT %MW20062.9 : BOOL; (* R366_1_M_I_RB_간섭무_10 *)
    R366_1_M_I_RB_간섭무_11 AT %MW20062.10 : BOOL; (* R366_1_M_I_RB_간섭무_11 *)
    R366_1_M_I_RB_간섭무_12 AT %MW20062.11 : BOOL; (* R366_1_M_I_RB_간섭무_12 *)
    R366_1_M_I_RB_간섭무_2 AT %MW20062.1 : BOOL; (* R366_1_M_I_RB_간섭무_2 *)
    R366_1_M_I_RB_간섭무_3 AT %MW20062.2 : BOOL; (* R366_1_M_I_RB_간섭무_3 *)
    R366_1_M_I_RB_간섭무_4 AT %MW20062.3 : BOOL; (* R366_1_M_I_RB_간섭무_4 *)
    R366_1_M_I_RB_간섭무_5 AT %MW20062.4 : BOOL; (* R366_1_M_I_RB_간섭무_5 *)
    R366_1_M_I_RB_간섭무_6 AT %MW20062.5 : BOOL; (* R366_1_M_I_RB_간섭무_6 *)
    R366_1_M_I_RB_간섭무_7 AT %MW20062.6 : BOOL; (* R366_1_M_I_RB_간섭무_7 *)
    R366_1_M_I_RB_간섭무_8 AT %MW20062.7 : BOOL; (* R366_1_M_I_RB_간섭무_8 *)
    R366_1_M_I_RB_간섭무_9 AT %MW20062.8 : BOOL; (* R366_1_M_I_RB_간섭무_9 *)
    R366_1_M_I_RB_비상정지 AT %MW20060.4 : BOOL; (* R366_1_M_I_RB_비상정지 *)
    R366_1_M_I_RB_운전준비 AT %MW20060.0 : BOOL; (* R366_1_M_I_RB_운전준비 *)
    R366_1_M_I_RB_원위치 AT %MW20060.3 : BOOL; (* R366_1_M_I_RB_원위치 *)
    R366_1_M_I_RB_이상 AT %MW20060.2 : BOOL; (* R366_1_M_I_RB_이상 *)
    R366_1_M_I_RB_자동 AT %MW20060.1 : BOOL; (* R366_1_M_I_RB_자동 *)
    R366_1_M_I_RB_최종작업완료 AT %MW20061.0 : BOOL; (* R366_1_M_I_RB_최종작업완료 *)
    R366_1_M_I_RB_프로그램_이상 AT %MW20060.6 : BOOL; (* R366_1_M_I_RB_프로그램_이상 *)
    R366_1_M_O_RB_1_CYCLE_SET AT %MW21060.3 : BOOL; (* R366_1_M_O_RB_1_CYCLE_SET *)
    R366_1_M_O_RB_1_CYCLE_리셋 AT %MW21060.4 : BOOL; (* R366_1_M_O_RB_1_CYCLE_리셋 *)
    R366_1_M_O_RB_1차_작업완료_리셋 AT %MW21062.0 : BOOL; (* R366_1_M_O_RB_1차_작업완료_리셋 *)
    R366_1_M_O_RB_2차_작업완료_리셋 AT %MW21062.1 : BOOL; (* R366_1_M_O_RB_2차_작업완료_리셋 *)
    R366_1_M_O_RB_2차_진입OK AT %MW21061.8 : BOOL; (* R366_1_M_O_RB_2차_진입OK *)
    R366_1_M_O_RB_3차_작업완료_리셋 AT %MW21062.2 : BOOL; (* R366_1_M_O_RB_3차_작업완료_리셋 *)
    R366_1_M_O_RB_3차_진입OK AT %MW21061.9 : BOOL; (* R366_1_M_O_RB_3차_진입OK *)
    R366_1_M_O_RB_4차_작업완료_리셋 AT %MW21062.3 : BOOL; (* R366_1_M_O_RB_4차_작업완료_리셋 *)
    R366_1_M_O_RB_4차_진입OK AT %MW21061.10 : BOOL; (* R366_1_M_O_RB_4차_진입OK *)
    R366_1_M_O_RB_5차_작업완료_리셋 AT %MW21062.4 : BOOL; (* R366_1_M_O_RB_5차_작업완료_리셋 *)
    R366_1_M_O_RB_5차_진입OK AT %MW21061.11 : BOOL; (* R366_1_M_O_RB_5차_진입OK *)
    R366_1_M_O_RB_6차_작업완료_리셋 AT %MW21062.5 : BOOL; (* R366_1_M_O_RB_6차_작업완료_리셋 *)
    R366_1_M_O_RB_6차_진입OK AT %MW21061.12 : BOOL; (* R366_1_M_O_RB_6차_진입OK *)
    R366_1_M_O_RB_7차_작업완료_리셋 AT %MW21062.6 : BOOL; (* R366_1_M_O_RB_7차_작업완료_리셋 *)
    R366_1_M_O_RB_7차_진입OK AT %MW21061.13 : BOOL; (* R366_1_M_O_RB_7차_진입OK *)
    R366_1_M_O_RB_ATD_OK AT %MW21060.6 : BOOL; (* R366_1_M_O_RB_ATD_OK *)
    R366_1_M_O_RB_PLT_10_진입OK AT %MW21063.10 : BOOL; (* R366_1_M_O_RB_PLT_10_진입OK *)
    R366_1_M_O_RB_PLT_11_진입OK AT %MW21063.11 : BOOL; (* R366_1_M_O_RB_PLT_11_진입OK *)
    R366_1_M_O_RB_PLT_12_진입OK AT %MW21063.12 : BOOL; (* R366_1_M_O_RB_PLT_12_진입OK *)
    R366_1_M_O_RB_PLT_1_진입OK AT %MW21063.1 : BOOL; (* R366_1_M_O_RB_PLT_1_진입OK *)
    R366_1_M_O_RB_PLT_2_진입OK AT %MW21063.2 : BOOL; (* R366_1_M_O_RB_PLT_2_진입OK *)
    R366_1_M_O_RB_PLT_3_진입OK AT %MW21063.3 : BOOL; (* R366_1_M_O_RB_PLT_3_진입OK *)
    R366_1_M_O_RB_PLT_4_진입OK AT %MW21063.4 : BOOL; (* R366_1_M_O_RB_PLT_4_진입OK *)
    R366_1_M_O_RB_PLT_5_진입OK AT %MW21063.5 : BOOL; (* R366_1_M_O_RB_PLT_5_진입OK *)
    R366_1_M_O_RB_PLT_6_진입OK AT %MW21063.6 : BOOL; (* R366_1_M_O_RB_PLT_6_진입OK *)
    R366_1_M_O_RB_PLT_7_진입OK AT %MW21063.7 : BOOL; (* R366_1_M_O_RB_PLT_7_진입OK *)
    R366_1_M_O_RB_PLT_8_진입OK AT %MW21063.8 : BOOL; (* R366_1_M_O_RB_PLT_8_진입OK *)
    R366_1_M_O_RB_PLT_9_진입OK AT %MW21063.9 : BOOL; (* R366_1_M_O_RB_PLT_9_진입OK *)
    R366_1_M_O_RB_PLT_카운터리셋_보조 AT %MW21060.10 : BOOL; (* R366_1_M_O_RB_PLT_카운터리셋_보조 *)
    R366_1_M_O_RB_PROG_NO AT %MW21064 : WORD;
    R366_1_M_O_RB_RESTART_OK AT %MW21060.2 : BOOL; (* R366_1_M_O_RB_RESTART_OK *)
    R366_1_M_O_RB_START_OK AT %MW21060.0 : BOOL; (* R366_1_M_O_RB_START_OK *)
    R366_1_M_O_RB_TEST_MODE_5000회 AT %MW21060.12 : BOOL; (* R366_1_M_O_RB_TEST_MODE_5000회 *)
    R366_1_M_O_RB_TIP_교체_시작 AT %MW21060.7 : BOOL; (* R366_1_M_O_RB_TIP_교체_시작 *)
    R366_1_M_O_RB_TIP_교체_완료 AT %MW21060.8 : BOOL; (* R366_1_M_O_RB_TIP_교체_완료 *)
    R366_1_M_O_RB_VIP_MODE AT %MW21060.11 : BOOL; (* R366_1_M_O_RB_VIP_MODE *)
    R366_1_M_O_RB_냉각수_차단_요청 AT %MW21060.9 : BOOL; (* R366_1_M_O_RB_냉각수_차단_요청 *)
    R366_1_M_O_RB_진입OK_AX차종 AT %MW21061.0 : BOOL; (* R366_1_M_O_RB_진입OK_AX차종 *)
    R366_1_M_O_RB_진입OK_B차종 AT %MW21061.1 : BOOL; (* R366_1_M_O_RB_진입OK_B차종 *)
    R366_1_M_O_RB_진입OK_C차종 AT %MW21061.2 : BOOL; (* R366_1_M_O_RB_진입OK_C차종 *)
    R366_1_M_O_RB_진입OK_D차종 AT %MW21061.3 : BOOL; (* R366_1_M_O_RB_진입OK_D차종 *)
    R366_1_M_O_RB_진입OK_E차종 AT %MW21061.4 : BOOL; (* R366_1_M_O_RB_진입OK_E차종 *)
    R366_1_M_O_RB_진입OK_F차종 AT %MW21061.5 : BOOL; (* R366_1_M_O_RB_진입OK_F차종 *)
    R366_1_M_O_RB_진입OK_G차종 AT %MW21061.6 : BOOL; (* R366_1_M_O_RB_진입OK_G차종 *)
    R366_1_M_O_RB_진입OK_H차종 AT %MW21061.7 : BOOL; (* R366_1_M_O_RB_진입OK_H차종 *)
    R366_1_M_O_RB_최종_작업완료_리셋 AT %MW21060.5 : BOOL; (* R366_1_M_O_RB_최종_작업완료_리셋 *)
    R366_1_M_O_RB_프로그램_OK AT %MW21060.1 : BOOL; (* R366_1_M_O_RB_프로그램_OK *)
    R366_1_O_RB_0_5S_통신_CHK AT %MW94063.14 : BOOL; (* R366_1_O_RB_0_5S_통신_CHK *)
    R366_1_O_RB_2차_진입OK AT %MW94061.8 : BOOL; (* R366_1_O_RB_2차_진입OK *)
    R366_1_O_RB_3차_진입OK AT %MW94061.9 : BOOL; (* R366_1_O_RB_3차_진입OK *)
    R366_1_O_RB_4차_진입OK AT %MW94061.10 : BOOL; (* R366_1_O_RB_4차_진입OK *)
    R366_1_O_RB_5차_진입OK AT %MW94061.11 : BOOL; (* R366_1_O_RB_5차_진입OK *)
    R366_1_O_RB_6차_진입OK AT %MW94061.12 : BOOL; (* R366_1_O_RB_6차_진입OK *)
    R366_1_O_RB_7차_진입OK AT %MW94061.13 : BOOL; (* R366_1_O_RB_7차_진입OK *)
    R366_1_O_RB_AX_1차_진입OK AT %MW94061.0 : BOOL; (* R366_1_O_RB_AX_1차_진입OK *)
    R366_1_O_RB_B_1차_진입OK AT %MW94061.1 : BOOL; (* R366_1_O_RB_B_1차_진입OK *)
    R366_1_O_RB_C_1차_진입OK AT %MW94061.2 : BOOL; (* R366_1_O_RB_C_1차_진입OK *)
    R366_1_O_RB_D_1차_진입OK AT %MW94061.3 : BOOL; (* R366_1_O_RB_D_1차_진입OK *)
    R366_1_O_RB_EACH_작업완료_리셋 AT %MW94060.14 : BOOL; (* R366_1_O_RB_EACH_작업완료_리셋 *)
    R366_1_O_RB_EXT_READY AT %MW94060.11 : BOOL; (* R366_1_O_RB_EXT_READY *)
    R366_1_O_RB_E_1차_진입OK AT %MW94061.4 : BOOL; (* R366_1_O_RB_E_1차_진입OK *)
    R366_1_O_RB_F_1차_진입OK AT %MW94061.5 : BOOL; (* R366_1_O_RB_F_1차_진입OK *)
    R366_1_O_RB_GATE_OPEN_NC AT %MW94063.11 : BOOL; (* R366_1_O_RB_GATE_OPEN_NC *)
    R366_1_O_RB_G_1차_진입OK AT %MW94061.6 : BOOL; (* R366_1_O_RB_G_1차_진입OK *)
    R366_1_O_RB_H_1차_진입OK AT %MW94061.7 : BOOL; (* R366_1_O_RB_H_1차_진입OK *)
    R366_1_O_RB_OUTPUT AT %MW94060 : ARRAY[0..3] OF WORD; (* R366_1_O_RB_OUTPUT *)
    R366_1_O_RB_PAUSE_NC AT %MW94060.13 : BOOL; (* R366_1_O_RB_PAUSE_NC *)
    R366_1_O_RB_PLT10_진입OK AT %MW94062.9 : BOOL; (* R366_1_O_RB_PLT10_진입OK *)
    R366_1_O_RB_PLT11_진입OK AT %MW94062.10 : BOOL; (* R366_1_O_RB_PLT11_진입OK *)
    R366_1_O_RB_PLT12_진입OK AT %MW94062.11 : BOOL; (* R366_1_O_RB_PLT12_진입OK *)
    R366_1_O_RB_PLT1_진입OK AT %MW94062.0 : BOOL; (* R366_1_O_RB_PLT1_진입OK *)
    R366_1_O_RB_PLT2_진입OK AT %MW94062.1 : BOOL; (* R366_1_O_RB_PLT2_진입OK *)
    R366_1_O_RB_PLT3_진입OK AT %MW94062.2 : BOOL; (* R366_1_O_RB_PLT3_진입OK *)
    R366_1_O_RB_PLT4_진입OK AT %MW94062.3 : BOOL; (* R366_1_O_RB_PLT4_진입OK *)
    R366_1_O_RB_PLT5_진입OK AT %MW94062.4 : BOOL; (* R366_1_O_RB_PLT5_진입OK *)
    R366_1_O_RB_PLT6_진입OK AT %MW94062.5 : BOOL; (* R366_1_O_RB_PLT6_진입OK *)
    R366_1_O_RB_PLT7_진입OK AT %MW94062.6 : BOOL; (* R366_1_O_RB_PLT7_진입OK *)
    R366_1_O_RB_PLT8_진입OK AT %MW94062.7 : BOOL; (* R366_1_O_RB_PLT8_진입OK *)
    R366_1_O_RB_PLT9_진입OK AT %MW94062.8 : BOOL; (* R366_1_O_RB_PLT9_진입OK *)
    R366_1_O_RB_PLT_카운터_리셋_요구 AT %MW94063.10 : BOOL; (* R366_1_O_RB_PLT_카운터_리셋_요구 *)
    R366_1_O_RB_PROG_선택1 AT %MW94060.0 : BOOL; (* R366_1_O_RB_PROG_선택1 *)
    R366_1_O_RB_PROG_선택128 AT %MW94060.7 : BOOL; (* R366_1_O_RB_PROG_선택128 *)
    R366_1_O_RB_PROG_선택16 AT %MW94060.4 : BOOL; (* R366_1_O_RB_PROG_선택16 *)
    R366_1_O_RB_PROG_선택2 AT %MW94060.1 : BOOL; (* R366_1_O_RB_PROG_선택2 *)
    R366_1_O_RB_PROG_선택32 AT %MW94060.5 : BOOL; (* R366_1_O_RB_PROG_선택32 *)
    R366_1_O_RB_PROG_선택4 AT %MW94060.2 : BOOL; (* R366_1_O_RB_PROG_선택4 *)
    R366_1_O_RB_PROG_선택64 AT %MW94060.6 : BOOL; (* R366_1_O_RB_PROG_선택64 *)
    R366_1_O_RB_PROG_선택8 AT %MW94060.3 : BOOL; (* R366_1_O_RB_PROG_선택8 *)
    R366_1_O_RB_SP_1_14 AT %MW94061.14 : BOOL; (* R366_1_O_RB_SP_1_14 *)
    R366_1_O_RB_SP_1_15 AT %MW94061.15 : BOOL; (* R366_1_O_RB_SP_1_15 *)
    R366_1_O_RB_SP_2_12 AT %MW94062.12 : BOOL; (* R366_1_O_RB_SP_2_12 *)
    R366_1_O_RB_SP_2_13 AT %MW94062.13 : BOOL; (* R366_1_O_RB_SP_2_13 *)
    R366_1_O_RB_SP_2_14 AT %MW94062.14 : BOOL; (* R366_1_O_RB_SP_2_14 *)
    R366_1_O_RB_SP_5000TH_ON AT %MW94062.15 : BOOL; (* R366_1_O_RB_SP_5000TH_ON *)
    R366_1_O_RB_TIP_CHANGE_END AT %MW94063.9 : BOOL; (* R366_1_O_RB_TIP_CHANGE_END *)
    R366_1_O_RB_TIP_CHANGE_START AT %MW94063.8 : BOOL; (* R366_1_O_RB_TIP_CHANGE_START *)
    R366_1_O_RB_TIP_DRESS_SATRT AT %MW94060.12 : BOOL; (* R366_1_O_RB_TIP_DRESS_SATRT *)
    R366_1_O_RB_VIP_MODE AT %MW94063.15 : BOOL; (* R366_1_O_RB_VIP_MODE *)
    R366_1_O_RB_기동 AT %MW94060.9 : BOOL; (* R366_1_O_RB_기동 *)
    R366_1_O_RB_냉각수차단 AT %MW94060.15 : BOOL; (* R366_1_O_RB_냉각수차단 *)
    R366_1_O_RB_부저정지 AT %MW94063.13 : BOOL; (* R366_1_O_RB_부저정지 *)
    R366_1_O_RB_비상정지_NC AT %MW94063.12 : BOOL; (* R366_1_O_RB_비상정지_NC *)
    R366_1_O_RB_상호인터록_INT1 AT %MW94063.0 : BOOL; (* R366_1_O_RB_상호인터록_INT1 *)
    R366_1_O_RB_상호인터록_INT2 AT %MW94063.1 : BOOL; (* R366_1_O_RB_상호인터록_INT2 *)
    R366_1_O_RB_상호인터록_INT3 AT %MW94063.2 : BOOL; (* R366_1_O_RB_상호인터록_INT3 *)
    R366_1_O_RB_상호인터록_INT4 AT %MW94063.3 : BOOL; (* R366_1_O_RB_상호인터록_INT4 *)
    R366_1_O_RB_상호인터록_INT5 AT %MW94063.4 : BOOL; (* R366_1_O_RB_상호인터록_INT5 *)
    R366_1_O_RB_상호인터록_INT6 AT %MW94063.5 : BOOL; (* R366_1_O_RB_상호인터록_INT6 *)
    R366_1_O_RB_상호인터록_INT7 AT %MW94063.6 : BOOL; (* R366_1_O_RB_상호인터록_INT7 *)
    R366_1_O_RB_상호인터록_INT8 AT %MW94063.7 : BOOL; (* R366_1_O_RB_상호인터록_INT8 *)
    R366_1_O_RB_이상_리셋 AT %MW94060.10 : BOOL; (* R366_1_O_RB_이상_리셋 *)
    R366_1_O_RB_작업완료_리셋 AT %MW94060.8 : BOOL; (* R366_1_O_RB_작업완료_리셋 *)
    R368_1_I_RB_0_5_COMM_CHK AT %MW84073.14 : BOOL; (* R368_1_I_RB_0_5_COMM_CHK *)
    R368_1_I_RB_10차_간섭무 AT %MW84071.9 : BOOL; (* R368_1_I_RB_10차_간섭무 *)
    R368_1_I_RB_11차_간섭무 AT %MW84071.10 : BOOL; (* R368_1_I_RB_11차_간섭무 *)
    R368_1_I_RB_12차_간섭무 AT %MW84071.11 : BOOL; (* R368_1_I_RB_12차_간섭무 *)
    R368_1_I_RB_1차_간섭무 AT %MW84071.0 : BOOL; (* R368_1_I_RB_1차_간섭무 *)
    R368_1_I_RB_1차_작업완료 AT %MW84070.9 : BOOL; (* R368_1_I_RB_1차_작업완료 *)
    R368_1_I_RB_2차_간섭무 AT %MW84071.1 : BOOL; (* R368_1_I_RB_2차_간섭무 *)
    R368_1_I_RB_2차_작업완료 AT %MW84070.10 : BOOL; (* R368_1_I_RB_2차_작업완료 *)
    R368_1_I_RB_3차_간섭무 AT %MW84071.2 : BOOL; (* R368_1_I_RB_3차_간섭무 *)
    R368_1_I_RB_3차_작업완료 AT %MW84070.11 : BOOL; (* R368_1_I_RB_3차_작업완료 *)
    R368_1_I_RB_4차_간섭무 AT %MW84071.3 : BOOL; (* R368_1_I_RB_4차_간섭무 *)
    R368_1_I_RB_4차_작업완료 AT %MW84070.12 : BOOL; (* R368_1_I_RB_4차_작업완료 *)
    R368_1_I_RB_5차_간섭무 AT %MW84071.4 : BOOL; (* R368_1_I_RB_5차_간섭무 *)
    R368_1_I_RB_5차_작업완료 AT %MW84070.13 : BOOL; (* R368_1_I_RB_5차_작업완료 *)
    R368_1_I_RB_6차_간섭무 AT %MW84071.5 : BOOL; (* R368_1_I_RB_6차_간섭무 *)
    R368_1_I_RB_6차_작업완료 AT %MW84070.14 : BOOL; (* R368_1_I_RB_6차_작업완료 *)
    R368_1_I_RB_7차_간섭무 AT %MW84071.6 : BOOL; (* R368_1_I_RB_7차_간섭무 *)
    R368_1_I_RB_7차_작업완료 AT %MW84070.15 : BOOL; (* R368_1_I_RB_7차_작업완료 *)
    R368_1_I_RB_8차_간섭무 AT %MW84071.7 : BOOL; (* R368_1_I_RB_8차_간섭무 *)
    R368_1_I_RB_9차_간섭무 AT %MW84071.8 : BOOL; (* R368_1_I_RB_9차_간섭무 *)
    R368_1_I_RB_AB_NORMAL_선택 AT %MW84070.6 : BOOL; (* R368_1_I_RB_AB_NORMAL_선택 *)
    R368_1_I_RB_GUN1_FIXED_TIP AT %MW84077 : WORD; (* R368_1_I_RB_GUN1_FIXED_TIP *)
    R368_1_I_RB_GUN1_MOVING_TIP AT %MW84076 : WORD; (* R368_1_I_RB_GUN1_MOVING_TIP *)
    R368_1_I_RB_GUN2_FIXED_TIP AT %MW84079 : WORD; (* R368_1_I_RB_GUN2_FIXED_TIP *)
    R368_1_I_RB_GUN2_MOVING_TIP AT %MW84078 : WORD; (* R368_1_I_RB_GUN2_MOVING_TIP *)
    R368_1_I_RB_INPUT AT %MW84070 : ARRAY[0..3] OF WORD; (* R368_1_I_RB_INPUT *)
    R368_1_I_RB_LS_이상 AT %MW84072.11 : BOOL; (* R368_1_I_RB_LS_이상 *)
    R368_1_I_RB_MOTOR_MC_ON AT %MW84073.15 : BOOL; (* R368_1_I_RB_MOTOR_MC_ON *)
    R368_1_I_RB_PLT_UNLOAD_완료 AT %MW84073.11 : BOOL; (* R368_1_I_RB_PLT_UNLOAD_완료 *)
    R368_1_I_RB_PLT_최종UNLOAD_완료 AT %MW84073.12 : BOOL; (* R368_1_I_RB_PLT_최종UNLOAD_완료 *)
    R368_1_I_RB_PROG_ECHO_1 AT %MW84072.0 : BOOL; (* R368_1_I_RB_PROG_ECHO_1 *)
    R368_1_I_RB_PROG_ECHO_128 AT %MW84072.7 : BOOL; (* R368_1_I_RB_PROG_ECHO_128 *)
    R368_1_I_RB_PROG_ECHO_16 AT %MW84072.4 : BOOL; (* R368_1_I_RB_PROG_ECHO_16 *)
    R368_1_I_RB_PROG_ECHO_2 AT %MW84072.1 : BOOL; (* R368_1_I_RB_PROG_ECHO_2 *)
    R368_1_I_RB_PROG_ECHO_32 AT %MW84072.5 : BOOL; (* R368_1_I_RB_PROG_ECHO_32 *)
    R368_1_I_RB_PROG_ECHO_4 AT %MW84072.2 : BOOL; (* R368_1_I_RB_PROG_ECHO_4 *)
    R368_1_I_RB_PROG_ECHO_64 AT %MW84072.6 : BOOL; (* R368_1_I_RB_PROG_ECHO_64 *)
    R368_1_I_RB_PROG_ECHO_8 AT %MW84072.3 : BOOL; (* R368_1_I_RB_PROG_ECHO_8 *)
    R368_1_I_RB_SP3_8 AT %MW84073.8 : BOOL; (* R368_1_I_RB_SP3_8 *)
    R368_1_I_RB_SP3_9 AT %MW84073.9 : BOOL; (* R368_1_I_RB_SP3_9 *)
    R368_1_I_RB_SPARE_WORD_4 AT %MW84074 : WORD; (* R368_1_I_RB_SPARE_WORD_4 *)
    R368_1_I_RB_SP_1_12 AT %MW84071.12 : BOOL; (* R368_1_I_RB_SP_1_12 *)
    R368_1_I_RB_SP_1_13 AT %MW84071.13 : BOOL; (* R368_1_I_RB_SP_1_13 *)
    R368_1_I_RB_SP_1_14 AT %MW84071.14 : BOOL; (* R368_1_I_RB_SP_1_14 *)
    R368_1_I_RB_SP_1_15 AT %MW84071.15 : BOOL; (* R368_1_I_RB_SP_1_15 *)
    R368_1_I_RB_TC_이상 AT %MW84072.8 : BOOL; (* R368_1_I_RB_TC_이상 *)
    R368_1_I_RB_TIP_CHANGE AT %MW84073.13 : BOOL; (* R368_1_I_RB_TIP_CHANGE *)
    R368_1_I_RB_TIP_DRESSING AT %MW84070.7 : BOOL; (* R368_1_I_RB_TIP_DRESSING *)
    R368_1_I_RB__PLT_카운터리셋완료 AT %MW84073.10 : BOOL; (* R368_1_I_RB__PLT_카운터리셋완료 *)
    R368_1_I_RB_공기압_이상 AT %MW84072.9 : BOOL; (* R368_1_I_RB_공기압_이상 *)
    R368_1_I_RB_냉각수_이상 AT %MW84072.10 : BOOL; (* R368_1_I_RB_냉각수_이상 *)
    R368_1_I_RB_비상정지_NC AT %MW84070.8 : BOOL; (* R368_1_I_RB_비상정지_NC *)
    R368_1_I_RB_비전이상 AT %MW84072.14 : BOOL; (* R368_1_I_RB_비전이상 *)
    R368_1_I_RB_상호인터록_INT1 AT %MW84073.0 : BOOL; (* R368_1_I_RB_상호인터록_INT1 *)
    R368_1_I_RB_상호인터록_INT2 AT %MW84073.1 : BOOL; (* R368_1_I_RB_상호인터록_INT2 *)
    R368_1_I_RB_상호인터록_INT3 AT %MW84073.2 : BOOL; (* R368_1_I_RB_상호인터록_INT3 *)
    R368_1_I_RB_상호인터록_INT4 AT %MW84073.3 : BOOL; (* R368_1_I_RB_상호인터록_INT4 *)
    R368_1_I_RB_상호인터록_INT5 AT %MW84073.4 : BOOL; (* R368_1_I_RB_상호인터록_INT5 *)
    R368_1_I_RB_상호인터록_INT6 AT %MW84073.5 : BOOL; (* R368_1_I_RB_상호인터록_INT6 *)
    R368_1_I_RB_상호인터록_INT7 AT %MW84073.6 : BOOL; (* R368_1_I_RB_상호인터록_INT7 *)
    R368_1_I_RB_상호인터록_INT8 AT %MW84073.7 : BOOL; (* R368_1_I_RB_상호인터록_INT8 *)
    R368_1_I_RB_실러이상 AT %MW84072.13 : BOOL; (* R368_1_I_RB_실러이상 *)
    R368_1_I_RB_용접카운터이상 AT %MW84072.15 : BOOL; (* R368_1_I_RB_용접카운터이상 *)
    R368_1_I_RB_용접타점수 AT %MW84075 : WORD; (* R368_1_I_RB_용접타점수 *)
    R368_1_I_RB_운전준비 AT %MW84070.3 : BOOL; (* R368_1_I_RB_운전준비 *)
    R368_1_I_RB_원위치 AT %MW84070.0 : BOOL; (* R368_1_I_RB_원위치 *)
    R368_1_I_RB_이상리셋 AT %MW84070.2 : BOOL; (* R368_1_I_RB_이상리셋 *)
    R368_1_I_RB_자동 AT %MW84070.4 : BOOL; (* R368_1_I_RB_자동 *)
    R368_1_I_RB_자동기동 AT %MW84070.5 : BOOL; (* R368_1_I_RB_자동기동 *)
    R368_1_I_RB_최종_작업완료 AT %MW84070.1 : BOOL; (* R368_1_I_RB_최종_작업완료 *)
    R368_1_I_RB_통신이상 AT %MW84072.12 : BOOL; (* R368_1_I_RB_통신이상 *)
    R368_1_M_I_RB_1차_작업완료 AT %MW20071.2 : BOOL; (* R368_1_M_I_RB_1차_작업완료 *)
    R368_1_M_I_RB_2차_작업완료 AT %MW20071.3 : BOOL; (* R368_1_M_I_RB_2차_작업완료 *)
    R368_1_M_I_RB_3차_작업완료 AT %MW20071.4 : BOOL; (* R368_1_M_I_RB_3차_작업완료 *)
    R368_1_M_I_RB_4차_작업완료 AT %MW20071.5 : BOOL; (* R368_1_M_I_RB_4차_작업완료 *)
    R368_1_M_I_RB_5차_작업완료 AT %MW20071.6 : BOOL; (* R368_1_M_I_RB_5차_작업완료 *)
    R368_1_M_I_RB_6차_작업완료 AT %MW20071.7 : BOOL; (* R368_1_M_I_RB_6차_작업완료 *)
    R368_1_M_I_RB_7차_작업완료 AT %MW20071.8 : BOOL; (* R368_1_M_I_RB_7차_작업완료 *)
    R368_1_M_I_RB_PAUSE_보조 AT %MW20070.5 : BOOL; (* R368_1_M_I_RB_PAUSE_보조 *)
    R368_1_M_I_RB_PLC_RUN_CHK_이상 AT %MW20070.7 : BOOL; (* R368_1_M_I_RB_PLC_RUN_CHK_이상 *)
    R368_1_M_I_RB_간섭무_1 AT %MW20072.0 : BOOL; (* R368_1_M_I_RB_간섭무_1 *)
    R368_1_M_I_RB_간섭무_10 AT %MW20072.9 : BOOL; (* R368_1_M_I_RB_간섭무_10 *)
    R368_1_M_I_RB_간섭무_11 AT %MW20072.10 : BOOL; (* R368_1_M_I_RB_간섭무_11 *)
    R368_1_M_I_RB_간섭무_12 AT %MW20072.11 : BOOL; (* R368_1_M_I_RB_간섭무_12 *)
    R368_1_M_I_RB_간섭무_2 AT %MW20072.1 : BOOL; (* R368_1_M_I_RB_간섭무_2 *)
    R368_1_M_I_RB_간섭무_3 AT %MW20072.2 : BOOL; (* R368_1_M_I_RB_간섭무_3 *)
    R368_1_M_I_RB_간섭무_4 AT %MW20072.3 : BOOL; (* R368_1_M_I_RB_간섭무_4 *)
    R368_1_M_I_RB_간섭무_5 AT %MW20072.4 : BOOL; (* R368_1_M_I_RB_간섭무_5 *)
    R368_1_M_I_RB_간섭무_6 AT %MW20072.5 : BOOL; (* R368_1_M_I_RB_간섭무_6 *)
    R368_1_M_I_RB_간섭무_7 AT %MW20072.6 : BOOL; (* R368_1_M_I_RB_간섭무_7 *)
    R368_1_M_I_RB_간섭무_8 AT %MW20072.7 : BOOL; (* R368_1_M_I_RB_간섭무_8 *)
    R368_1_M_I_RB_간섭무_9 AT %MW20072.8 : BOOL; (* R368_1_M_I_RB_간섭무_9 *)
    R368_1_M_I_RB_비상정지 AT %MW20070.4 : BOOL; (* R368_1_M_I_RB_비상정지 *)
    R368_1_M_I_RB_운전준비 AT %MW20070.0 : BOOL; (* R368_1_M_I_RB_운전준비 *)
    R368_1_M_I_RB_원위치 AT %MW20070.3 : BOOL; (* R368_1_M_I_RB_원위치 *)
    R368_1_M_I_RB_이상 AT %MW20070.2 : BOOL; (* R368_1_M_I_RB_이상 *)
    R368_1_M_I_RB_자동 AT %MW20070.1 : BOOL; (* R368_1_M_I_RB_자동 *)
    R368_1_M_I_RB_최종작업완료 AT %MW20071.0 : BOOL; (* R368_1_M_I_RB_최종작업완료 *)
    R368_1_M_I_RB_프로그램_이상 AT %MW20070.6 : BOOL; (* R368_1_M_I_RB_프로그램_이상 *)
    R368_1_M_O_RB_1_CYCLE_SET AT %MW21070.3 : BOOL; (* R368_1_M_O_RB_1_CYCLE_SET *)
    R368_1_M_O_RB_1_CYCLE_리셋 AT %MW21070.4 : BOOL; (* R368_1_M_O_RB_1_CYCLE_리셋 *)
    R368_1_M_O_RB_1차_작업완료_리셋 AT %MW21072.0 : BOOL; (* R368_1_M_O_RB_1차_작업완료_리셋 *)
    R368_1_M_O_RB_2차_작업완료_리셋 AT %MW21072.1 : BOOL; (* R368_1_M_O_RB_2차_작업완료_리셋 *)
    R368_1_M_O_RB_2차_진입OK AT %MW21071.8 : BOOL; (* R368_1_M_O_RB_2차_진입OK *)
    R368_1_M_O_RB_3차_작업완료_리셋 AT %MW21072.2 : BOOL; (* R368_1_M_O_RB_3차_작업완료_리셋 *)
    R368_1_M_O_RB_3차_진입OK AT %MW21071.9 : BOOL; (* R368_1_M_O_RB_3차_진입OK *)
    R368_1_M_O_RB_4차_작업완료_리셋 AT %MW21072.3 : BOOL; (* R368_1_M_O_RB_4차_작업완료_리셋 *)
    R368_1_M_O_RB_4차_진입OK AT %MW21071.10 : BOOL; (* R368_1_M_O_RB_4차_진입OK *)
    R368_1_M_O_RB_5차_작업완료_리셋 AT %MW21072.4 : BOOL; (* R368_1_M_O_RB_5차_작업완료_리셋 *)
    R368_1_M_O_RB_5차_진입OK AT %MW21071.11 : BOOL; (* R368_1_M_O_RB_5차_진입OK *)
    R368_1_M_O_RB_6차_작업완료_리셋 AT %MW21072.5 : BOOL; (* R368_1_M_O_RB_6차_작업완료_리셋 *)
    R368_1_M_O_RB_6차_진입OK AT %MW21071.12 : BOOL; (* R368_1_M_O_RB_6차_진입OK *)
    R368_1_M_O_RB_7차_작업완료_리셋 AT %MW21072.6 : BOOL; (* R368_1_M_O_RB_7차_작업완료_리셋 *)
    R368_1_M_O_RB_7차_진입OK AT %MW21071.13 : BOOL; (* R368_1_M_O_RB_7차_진입OK *)
    R368_1_M_O_RB_ATD_OK AT %MW21070.6 : BOOL; (* R368_1_M_O_RB_ATD_OK *)
    R368_1_M_O_RB_PLT_10_진입OK AT %MW21073.10 : BOOL; (* R368_1_M_O_RB_PLT_10_진입OK *)
    R368_1_M_O_RB_PLT_11_진입OK AT %MW21073.11 : BOOL; (* R368_1_M_O_RB_PLT_11_진입OK *)
    R368_1_M_O_RB_PLT_12_진입OK AT %MW21073.12 : BOOL; (* R368_1_M_O_RB_PLT_12_진입OK *)
    R368_1_M_O_RB_PLT_1_진입OK AT %MW21073.1 : BOOL; (* R368_1_M_O_RB_PLT_1_진입OK *)
    R368_1_M_O_RB_PLT_2_진입OK AT %MW21073.2 : BOOL; (* R368_1_M_O_RB_PLT_2_진입OK *)
    R368_1_M_O_RB_PLT_3_진입OK AT %MW21073.3 : BOOL; (* R368_1_M_O_RB_PLT_3_진입OK *)
    R368_1_M_O_RB_PLT_4_진입OK AT %MW21073.4 : BOOL; (* R368_1_M_O_RB_PLT_4_진입OK *)
    R368_1_M_O_RB_PLT_5_진입OK AT %MW21073.5 : BOOL; (* R368_1_M_O_RB_PLT_5_진입OK *)
    R368_1_M_O_RB_PLT_6_진입OK AT %MW21073.6 : BOOL; (* R368_1_M_O_RB_PLT_6_진입OK *)
    R368_1_M_O_RB_PLT_7_진입OK AT %MW21073.7 : BOOL; (* R368_1_M_O_RB_PLT_7_진입OK *)
    R368_1_M_O_RB_PLT_8_진입OK AT %MW21073.8 : BOOL; (* R368_1_M_O_RB_PLT_8_진입OK *)
    R368_1_M_O_RB_PLT_9_진입OK AT %MW21073.9 : BOOL; (* R368_1_M_O_RB_PLT_9_진입OK *)
    R368_1_M_O_RB_PLT_카운터리셋_보조 AT %MW21070.10 : BOOL; (* R368_1_M_O_RB_PLT_카운터리셋_보조 *)
    R368_1_M_O_RB_PROG_NO AT %MW21074 : WORD;
    R368_1_M_O_RB_RESTART_OK AT %MW21070.2 : BOOL; (* R368_1_M_O_RB_RESTART_OK *)
    R368_1_M_O_RB_START_OK AT %MW21070.0 : BOOL; (* R368_1_M_O_RB_START_OK *)
    R368_1_M_O_RB_TEST_MODE_5000회 AT %MW21070.12 : BOOL; (* R368_1_M_O_RB_TEST_MODE_5000회 *)
    R368_1_M_O_RB_TIP_교체_시작 AT %MW21070.7 : BOOL; (* R368_1_M_O_RB_TIP_교체_시작 *)
    R368_1_M_O_RB_TIP_교체_완료 AT %MW21070.8 : BOOL; (* R368_1_M_O_RB_TIP_교체_완료 *)
    R368_1_M_O_RB_VIP_MODE AT %MW21070.11 : BOOL; (* R368_1_M_O_RB_VIP_MODE *)
    R368_1_M_O_RB_냉각수_차단_요청 AT %MW21070.9 : BOOL; (* R368_1_M_O_RB_냉각수_차단_요청 *)
    R368_1_M_O_RB_진입OK_AX차종 AT %MW21071.0 : BOOL; (* R368_1_M_O_RB_진입OK_AX차종 *)
    R368_1_M_O_RB_진입OK_B차종 AT %MW21071.1 : BOOL; (* R368_1_M_O_RB_진입OK_B차종 *)
    R368_1_M_O_RB_진입OK_C차종 AT %MW21071.2 : BOOL; (* R368_1_M_O_RB_진입OK_C차종 *)
    R368_1_M_O_RB_진입OK_D차종 AT %MW21071.3 : BOOL; (* R368_1_M_O_RB_진입OK_D차종 *)
    R368_1_M_O_RB_진입OK_E차종 AT %MW21071.4 : BOOL; (* R368_1_M_O_RB_진입OK_E차종 *)
    R368_1_M_O_RB_진입OK_F차종 AT %MW21071.5 : BOOL; (* R368_1_M_O_RB_진입OK_F차종 *)
    R368_1_M_O_RB_진입OK_G차종 AT %MW21071.6 : BOOL; (* R368_1_M_O_RB_진입OK_G차종 *)
    R368_1_M_O_RB_진입OK_H차종 AT %MW21071.7 : BOOL; (* R368_1_M_O_RB_진입OK_H차종 *)
    R368_1_M_O_RB_최종_작업완료_리셋 AT %MW21070.5 : BOOL; (* R368_1_M_O_RB_최종_작업완료_리셋 *)
    R368_1_M_O_RB_프로그램_OK AT %MW21070.1 : BOOL; (* R368_1_M_O_RB_프로그램_OK *)
    R368_1_O_RB_0_5S_통신_CHK AT %MW94073.14 : BOOL; (* R368_1_O_RB_0_5S_통신_CHK *)
    R368_1_O_RB_2차_진입OK AT %MW94071.8 : BOOL; (* R368_1_O_RB_2차_진입OK *)
    R368_1_O_RB_3차_진입OK AT %MW94071.9 : BOOL; (* R368_1_O_RB_3차_진입OK *)
    R368_1_O_RB_4차_진입OK AT %MW94071.10 : BOOL; (* R368_1_O_RB_4차_진입OK *)
    R368_1_O_RB_5차_진입OK AT %MW94071.11 : BOOL; (* R368_1_O_RB_5차_진입OK *)
    R368_1_O_RB_6차_진입OK AT %MW94071.12 : BOOL; (* R368_1_O_RB_6차_진입OK *)
    R368_1_O_RB_7차_진입OK AT %MW94071.13 : BOOL; (* R368_1_O_RB_7차_진입OK *)
    R368_1_O_RB_AX_1차_진입OK AT %MW94071.0 : BOOL; (* R368_1_O_RB_AX_1차_진입OK *)
    R368_1_O_RB_B_1차_진입OK AT %MW94071.1 : BOOL; (* R368_1_O_RB_B_1차_진입OK *)
    R368_1_O_RB_C_1차_진입OK AT %MW94071.2 : BOOL; (* R368_1_O_RB_C_1차_진입OK *)
    R368_1_O_RB_D_1차_진입OK AT %MW94071.3 : BOOL; (* R368_1_O_RB_D_1차_진입OK *)
    R368_1_O_RB_EACH_작업완료_리셋 AT %MW94070.14 : BOOL; (* R368_1_O_RB_EACH_작업완료_리셋 *)
    R368_1_O_RB_EXT_READY AT %MW94070.11 : BOOL; (* R368_1_O_RB_EXT_READY *)
    R368_1_O_RB_E_1차_진입OK AT %MW94071.4 : BOOL; (* R368_1_O_RB_E_1차_진입OK *)
    R368_1_O_RB_F_1차_진입OK AT %MW94071.5 : BOOL; (* R368_1_O_RB_F_1차_진입OK *)
    R368_1_O_RB_GATE_OPEN_NC AT %MW94073.11 : BOOL; (* R368_1_O_RB_GATE_OPEN_NC *)
    R368_1_O_RB_G_1차_진입OK AT %MW94071.6 : BOOL; (* R368_1_O_RB_G_1차_진입OK *)
    R368_1_O_RB_H_1차_진입OK AT %MW94071.7 : BOOL; (* R368_1_O_RB_H_1차_진입OK *)
    R368_1_O_RB_OUTPUT AT %MW94070 : ARRAY[0..3] OF WORD; (* R368_1_O_RB_OUTPUT *)
    R368_1_O_RB_PAUSE_NC AT %MW94070.13 : BOOL; (* R368_1_O_RB_PAUSE_NC *)
    R368_1_O_RB_PLT10_진입OK AT %MW94072.9 : BOOL; (* R368_1_O_RB_PLT10_진입OK *)
    R368_1_O_RB_PLT11_진입OK AT %MW94072.10 : BOOL; (* R368_1_O_RB_PLT11_진입OK *)
    R368_1_O_RB_PLT12_진입OK AT %MW94072.11 : BOOL; (* R368_1_O_RB_PLT12_진입OK *)
    R368_1_O_RB_PLT1_진입OK AT %MW94072.0 : BOOL; (* R368_1_O_RB_PLT1_진입OK *)
    R368_1_O_RB_PLT2_진입OK AT %MW94072.1 : BOOL; (* R368_1_O_RB_PLT2_진입OK *)
    R368_1_O_RB_PLT3_진입OK AT %MW94072.2 : BOOL; (* R368_1_O_RB_PLT3_진입OK *)
    R368_1_O_RB_PLT4_진입OK AT %MW94072.3 : BOOL; (* R368_1_O_RB_PLT4_진입OK *)
    R368_1_O_RB_PLT5_진입OK AT %MW94072.4 : BOOL; (* R368_1_O_RB_PLT5_진입OK *)
    R368_1_O_RB_PLT6_진입OK AT %MW94072.5 : BOOL; (* R368_1_O_RB_PLT6_진입OK *)
    R368_1_O_RB_PLT7_진입OK AT %MW94072.6 : BOOL; (* R368_1_O_RB_PLT7_진입OK *)
    R368_1_O_RB_PLT8_진입OK AT %MW94072.7 : BOOL; (* R368_1_O_RB_PLT8_진입OK *)
    R368_1_O_RB_PLT9_진입OK AT %MW94072.8 : BOOL; (* R368_1_O_RB_PLT9_진입OK *)
    R368_1_O_RB_PLT_카운터_리셋_요구 AT %MW94073.10 : BOOL; (* R368_1_O_RB_PLT_카운터_리셋_요구 *)
    R368_1_O_RB_PROG_선택1 AT %MW94070.0 : BOOL; (* R368_1_O_RB_PROG_선택1 *)
    R368_1_O_RB_PROG_선택128 AT %MW94070.7 : BOOL; (* R368_1_O_RB_PROG_선택128 *)
    R368_1_O_RB_PROG_선택16 AT %MW94070.4 : BOOL; (* R368_1_O_RB_PROG_선택16 *)
    R368_1_O_RB_PROG_선택2 AT %MW94070.1 : BOOL; (* R368_1_O_RB_PROG_선택2 *)
    R368_1_O_RB_PROG_선택32 AT %MW94070.5 : BOOL; (* R368_1_O_RB_PROG_선택32 *)
    R368_1_O_RB_PROG_선택4 AT %MW94070.2 : BOOL; (* R368_1_O_RB_PROG_선택4 *)
    R368_1_O_RB_PROG_선택64 AT %MW94070.6 : BOOL; (* R368_1_O_RB_PROG_선택64 *)
    R368_1_O_RB_PROG_선택8 AT %MW94070.3 : BOOL; (* R368_1_O_RB_PROG_선택8 *)
    R368_1_O_RB_SP_1_14 AT %MW94071.14 : BOOL; (* R368_1_O_RB_SP_1_14 *)
    R368_1_O_RB_SP_1_15 AT %MW94071.15 : BOOL; (* R368_1_O_RB_SP_1_15 *)
    R368_1_O_RB_SP_2_12 AT %MW94072.12 : BOOL; (* R368_1_O_RB_SP_2_12 *)
    R368_1_O_RB_SP_2_13 AT %MW94072.13 : BOOL; (* R368_1_O_RB_SP_2_13 *)
    R368_1_O_RB_SP_2_14 AT %MW94072.14 : BOOL; (* R368_1_O_RB_SP_2_14 *)
    R368_1_O_RB_SP_5000TH_ON AT %MW94072.15 : BOOL; (* R368_1_O_RB_SP_5000TH_ON *)
    R368_1_O_RB_TIP_CHANGE_END AT %MW94073.9 : BOOL; (* R368_1_O_RB_TIP_CHANGE_END *)
    R368_1_O_RB_TIP_CHANGE_START AT %MW94073.8 : BOOL; (* R368_1_O_RB_TIP_CHANGE_START *)
    R368_1_O_RB_TIP_DRESS_SATRT AT %MW94070.12 : BOOL; (* R368_1_O_RB_TIP_DRESS_SATRT *)
    R368_1_O_RB_VIP_MODE AT %MW94073.15 : BOOL; (* R368_1_O_RB_VIP_MODE *)
    R368_1_O_RB_기동 AT %MW94070.9 : BOOL; (* R368_1_O_RB_기동 *)
    R368_1_O_RB_냉각수차단 AT %MW94070.15 : BOOL; (* R368_1_O_RB_냉각수차단 *)
    R368_1_O_RB_부저정지 AT %MW94073.13 : BOOL; (* R368_1_O_RB_부저정지 *)
    R368_1_O_RB_비상정지_NC AT %MW94073.12 : BOOL; (* R368_1_O_RB_비상정지_NC *)
    R368_1_O_RB_상호인터록_INT1 AT %MW94073.0 : BOOL; (* R368_1_O_RB_상호인터록_INT1 *)
    R368_1_O_RB_상호인터록_INT2 AT %MW94073.1 : BOOL; (* R368_1_O_RB_상호인터록_INT2 *)
    R368_1_O_RB_상호인터록_INT3 AT %MW94073.2 : BOOL; (* R368_1_O_RB_상호인터록_INT3 *)
    R368_1_O_RB_상호인터록_INT4 AT %MW94073.3 : BOOL; (* R368_1_O_RB_상호인터록_INT4 *)
    R368_1_O_RB_상호인터록_INT5 AT %MW94073.4 : BOOL; (* R368_1_O_RB_상호인터록_INT5 *)
    R368_1_O_RB_상호인터록_INT6 AT %MW94073.5 : BOOL; (* R368_1_O_RB_상호인터록_INT6 *)
    R368_1_O_RB_상호인터록_INT7 AT %MW94073.6 : BOOL; (* R368_1_O_RB_상호인터록_INT7 *)
    R368_1_O_RB_상호인터록_INT8 AT %MW94073.7 : BOOL; (* R368_1_O_RB_상호인터록_INT8 *)
    R368_1_O_RB_이상_리셋 AT %MW94070.10 : BOOL; (* R368_1_O_RB_이상_리셋 *)
    R368_1_O_RB_작업완료_리셋 AT %MW94070.8 : BOOL; (* R368_1_O_RB_작업완료_리셋 *)
    R369_1_I_RB_0_5_COMM_CHK AT %MW84083.14 : BOOL; (* R369_1_I_RB_0_5_COMM_CHK *)
    R369_1_I_RB_10차_간섭무 AT %MW84081.9 : BOOL; (* R369_1_I_RB_10차_간섭무 *)
    R369_1_I_RB_11차_간섭무 AT %MW84081.10 : BOOL; (* R369_1_I_RB_11차_간섭무 *)
    R369_1_I_RB_12차_간섭무 AT %MW84081.11 : BOOL; (* R369_1_I_RB_12차_간섭무 *)
    R369_1_I_RB_1차_간섭무 AT %MW84081.0 : BOOL; (* R369_1_I_RB_1차_간섭무 *)
    R369_1_I_RB_1차_작업완료 AT %MW84080.9 : BOOL; (* R369_1_I_RB_1차_작업완료 *)
    R369_1_I_RB_2차_간섭무 AT %MW84081.1 : BOOL; (* R369_1_I_RB_2차_간섭무 *)
    R369_1_I_RB_2차_작업완료 AT %MW84080.10 : BOOL; (* R369_1_I_RB_2차_작업완료 *)
    R369_1_I_RB_3차_간섭무 AT %MW84081.2 : BOOL; (* R369_1_I_RB_3차_간섭무 *)
    R369_1_I_RB_3차_작업완료 AT %MW84080.11 : BOOL; (* R369_1_I_RB_3차_작업완료 *)
    R369_1_I_RB_4차_간섭무 AT %MW84081.3 : BOOL; (* R369_1_I_RB_4차_간섭무 *)
    R369_1_I_RB_4차_작업완료 AT %MW84080.12 : BOOL; (* R369_1_I_RB_4차_작업완료 *)
    R369_1_I_RB_5차_간섭무 AT %MW84081.4 : BOOL; (* R369_1_I_RB_5차_간섭무 *)
    R369_1_I_RB_5차_작업완료 AT %MW84080.13 : BOOL; (* R369_1_I_RB_5차_작업완료 *)
    R369_1_I_RB_6차_간섭무 AT %MW84081.5 : BOOL; (* R369_1_I_RB_6차_간섭무 *)
    R369_1_I_RB_6차_작업완료 AT %MW84080.14 : BOOL; (* R369_1_I_RB_6차_작업완료 *)
    R369_1_I_RB_7차_간섭무 AT %MW84081.6 : BOOL; (* R369_1_I_RB_7차_간섭무 *)
    R369_1_I_RB_7차_작업완료 AT %MW84080.15 : BOOL; (* R369_1_I_RB_7차_작업완료 *)
    R369_1_I_RB_8차_간섭무 AT %MW84081.7 : BOOL; (* R369_1_I_RB_8차_간섭무 *)
    R369_1_I_RB_9차_간섭무 AT %MW84081.8 : BOOL; (* R369_1_I_RB_9차_간섭무 *)
    R369_1_I_RB_AB_NORMAL_선택 AT %MW84080.6 : BOOL; (* R369_1_I_RB_AB_NORMAL_선택 *)
    R369_1_I_RB_GUN1_FIXED_TIP AT %MW84087 : WORD; (* R369_1_I_RB_GUN1_FIXED_TIP *)
    R369_1_I_RB_GUN1_MOVING_TIP AT %MW84086 : WORD; (* R369_1_I_RB_GUN1_MOVING_TIP *)
    R369_1_I_RB_GUN2_FIXED_TIP AT %MW84089 : WORD; (* R369_1_I_RB_GUN2_FIXED_TIP *)
    R369_1_I_RB_GUN2_MOVING_TIP AT %MW84088 : WORD; (* R369_1_I_RB_GUN2_MOVING_TIP *)
    R369_1_I_RB_INPUT AT %MW84080 : ARRAY[0..3] OF WORD; (* R369_1_I_RB_INPUT *)
    R369_1_I_RB_LS_이상 AT %MW84082.11 : BOOL; (* R369_1_I_RB_LS_이상 *)
    R369_1_I_RB_MOTOR_MC_ON AT %MW84083.15 : BOOL; (* R369_1_I_RB_MOTOR_MC_ON *)
    R369_1_I_RB_PLT_UNLOAD_완료 AT %MW84083.11 : BOOL; (* R369_1_I_RB_PLT_UNLOAD_완료 *)
    R369_1_I_RB_PLT_최종UNLOAD_완료 AT %MW84083.12 : BOOL; (* R369_1_I_RB_PLT_최종UNLOAD_완료 *)
    R369_1_I_RB_PROG_ECHO_1 AT %MW84082.0 : BOOL; (* R369_1_I_RB_PROG_ECHO_1 *)
    R369_1_I_RB_PROG_ECHO_128 AT %MW84082.7 : BOOL; (* R369_1_I_RB_PROG_ECHO_128 *)
    R369_1_I_RB_PROG_ECHO_16 AT %MW84082.4 : BOOL; (* R369_1_I_RB_PROG_ECHO_16 *)
    R369_1_I_RB_PROG_ECHO_2 AT %MW84082.1 : BOOL; (* R369_1_I_RB_PROG_ECHO_2 *)
    R369_1_I_RB_PROG_ECHO_32 AT %MW84082.5 : BOOL; (* R369_1_I_RB_PROG_ECHO_32 *)
    R369_1_I_RB_PROG_ECHO_4 AT %MW84082.2 : BOOL; (* R369_1_I_RB_PROG_ECHO_4 *)
    R369_1_I_RB_PROG_ECHO_64 AT %MW84082.6 : BOOL; (* R369_1_I_RB_PROG_ECHO_64 *)
    R369_1_I_RB_PROG_ECHO_8 AT %MW84082.3 : BOOL; (* R369_1_I_RB_PROG_ECHO_8 *)
    R369_1_I_RB_SP3_8 AT %MW84083.8 : BOOL; (* R369_1_I_RB_SP3_8 *)
    R369_1_I_RB_SP3_9 AT %MW84083.9 : BOOL; (* R369_1_I_RB_SP3_9 *)
    R369_1_I_RB_SPARE_WORD_4 AT %MW84084 : WORD; (* R369_1_I_RB_SPARE_WORD_4 *)
    R369_1_I_RB_SP_1_12 AT %MW84081.12 : BOOL; (* R369_1_I_RB_SP_1_12 *)
    R369_1_I_RB_SP_1_13 AT %MW84081.13 : BOOL; (* R369_1_I_RB_SP_1_13 *)
    R369_1_I_RB_SP_1_14 AT %MW84081.14 : BOOL; (* R369_1_I_RB_SP_1_14 *)
    R369_1_I_RB_SP_1_15 AT %MW84081.15 : BOOL; (* R369_1_I_RB_SP_1_15 *)
    R369_1_I_RB_TC_이상 AT %MW84082.8 : BOOL; (* R369_1_I_RB_TC_이상 *)
    R369_1_I_RB_TIP_CHANGE AT %MW84083.13 : BOOL; (* R369_1_I_RB_TIP_CHANGE *)
    R369_1_I_RB_TIP_DRESSING AT %MW84080.7 : BOOL; (* R369_1_I_RB_TIP_DRESSING *)
    R369_1_I_RB__PLT_카운터리셋완료 AT %MW84083.10 : BOOL; (* R369_1_I_RB__PLT_카운터리셋완료 *)
    R369_1_I_RB_공기압_이상 AT %MW84082.9 : BOOL; (* R369_1_I_RB_공기압_이상 *)
    R369_1_I_RB_냉각수_이상 AT %MW84082.10 : BOOL; (* R369_1_I_RB_냉각수_이상 *)
    R369_1_I_RB_비상정지_NC AT %MW84080.8 : BOOL; (* R369_1_I_RB_비상정지_NC *)
    R369_1_I_RB_비전이상 AT %MW84082.14 : BOOL; (* R369_1_I_RB_비전이상 *)
    R369_1_I_RB_상호인터록_INT1 AT %MW84083.0 : BOOL; (* R369_1_I_RB_상호인터록_INT1 *)
    R369_1_I_RB_상호인터록_INT2 AT %MW84083.1 : BOOL; (* R369_1_I_RB_상호인터록_INT2 *)
    R369_1_I_RB_상호인터록_INT3 AT %MW84083.2 : BOOL; (* R369_1_I_RB_상호인터록_INT3 *)
    R369_1_I_RB_상호인터록_INT4 AT %MW84083.3 : BOOL; (* R369_1_I_RB_상호인터록_INT4 *)
    R369_1_I_RB_상호인터록_INT5 AT %MW84083.4 : BOOL; (* R369_1_I_RB_상호인터록_INT5 *)
    R369_1_I_RB_상호인터록_INT6 AT %MW84083.5 : BOOL; (* R369_1_I_RB_상호인터록_INT6 *)
    R369_1_I_RB_상호인터록_INT7 AT %MW84083.6 : BOOL; (* R369_1_I_RB_상호인터록_INT7 *)
    R369_1_I_RB_상호인터록_INT8 AT %MW84083.7 : BOOL; (* R369_1_I_RB_상호인터록_INT8 *)
    R369_1_I_RB_실러이상 AT %MW84082.13 : BOOL; (* R369_1_I_RB_실러이상 *)
    R369_1_I_RB_용접카운터이상 AT %MW84082.15 : BOOL; (* R369_1_I_RB_용접카운터이상 *)
    R369_1_I_RB_용접타점수 AT %MW84085 : WORD; (* R369_1_I_RB_용접타점수 *)
    R369_1_I_RB_운전준비 AT %MW84080.3 : BOOL; (* R369_1_I_RB_운전준비 *)
    R369_1_I_RB_원위치 AT %MW84080.0 : BOOL; (* R369_1_I_RB_원위치 *)
    R369_1_I_RB_이상리셋 AT %MW84080.2 : BOOL; (* R369_1_I_RB_이상리셋 *)
    R369_1_I_RB_자동 AT %MW84080.4 : BOOL; (* R369_1_I_RB_자동 *)
    R369_1_I_RB_자동기동 AT %MW84080.5 : BOOL; (* R369_1_I_RB_자동기동 *)
    R369_1_I_RB_최종_작업완료 AT %MW84080.1 : BOOL; (* R369_1_I_RB_최종_작업완료 *)
    R369_1_I_RB_통신이상 AT %MW84082.12 : BOOL; (* R369_1_I_RB_통신이상 *)
    R369_1_M_I_RB_1차_작업완료 AT %MW20081.2 : BOOL; (* R369_1_M_I_RB_1차_작업완료 *)
    R369_1_M_I_RB_2차_작업완료 AT %MW20081.3 : BOOL; (* R369_1_M_I_RB_2차_작업완료 *)
    R369_1_M_I_RB_3차_작업완료 AT %MW20081.4 : BOOL; (* R369_1_M_I_RB_3차_작업완료 *)
    R369_1_M_I_RB_4차_작업완료 AT %MW20081.5 : BOOL; (* R369_1_M_I_RB_4차_작업완료 *)
    R369_1_M_I_RB_5차_작업완료 AT %MW20081.6 : BOOL; (* R369_1_M_I_RB_5차_작업완료 *)
    R369_1_M_I_RB_6차_작업완료 AT %MW20081.7 : BOOL; (* R369_1_M_I_RB_6차_작업완료 *)
    R369_1_M_I_RB_7차_작업완료 AT %MW20081.8 : BOOL; (* R369_1_M_I_RB_7차_작업완료 *)
    R369_1_M_I_RB_PAUSE_보조 AT %MW20080.5 : BOOL; (* R369_1_M_I_RB_PAUSE_보조 *)
    R369_1_M_I_RB_PLC_RUN_CHK_이상 AT %MW20080.7 : BOOL; (* R369_1_M_I_RB_PLC_RUN_CHK_이상 *)
    R369_1_M_I_RB_간섭무_1 AT %MW20082.0 : BOOL; (* R369_1_M_I_RB_간섭무_1 *)
    R369_1_M_I_RB_간섭무_10 AT %MW20082.9 : BOOL; (* R369_1_M_I_RB_간섭무_10 *)
    R369_1_M_I_RB_간섭무_11 AT %MW20082.10 : BOOL; (* R369_1_M_I_RB_간섭무_11 *)
    R369_1_M_I_RB_간섭무_12 AT %MW20082.11 : BOOL; (* R369_1_M_I_RB_간섭무_12 *)
    R369_1_M_I_RB_간섭무_2 AT %MW20082.1 : BOOL; (* R369_1_M_I_RB_간섭무_2 *)
    R369_1_M_I_RB_간섭무_3 AT %MW20082.2 : BOOL; (* R369_1_M_I_RB_간섭무_3 *)
    R369_1_M_I_RB_간섭무_4 AT %MW20082.3 : BOOL; (* R369_1_M_I_RB_간섭무_4 *)
    R369_1_M_I_RB_간섭무_5 AT %MW20082.4 : BOOL; (* R369_1_M_I_RB_간섭무_5 *)
    R369_1_M_I_RB_간섭무_6 AT %MW20082.5 : BOOL; (* R369_1_M_I_RB_간섭무_6 *)
    R369_1_M_I_RB_간섭무_7 AT %MW20082.6 : BOOL; (* R369_1_M_I_RB_간섭무_7 *)
    R369_1_M_I_RB_간섭무_8 AT %MW20082.7 : BOOL; (* R369_1_M_I_RB_간섭무_8 *)
    R369_1_M_I_RB_간섭무_9 AT %MW20082.8 : BOOL; (* R369_1_M_I_RB_간섭무_9 *)
    R369_1_M_I_RB_비상정지 AT %MW20080.4 : BOOL; (* R369_1_M_I_RB_비상정지 *)
    R369_1_M_I_RB_운전준비 AT %MW20080.0 : BOOL; (* R369_1_M_I_RB_운전준비 *)
    R369_1_M_I_RB_원위치 AT %MW20080.3 : BOOL; (* R369_1_M_I_RB_원위치 *)
    R369_1_M_I_RB_이상 AT %MW20080.2 : BOOL; (* R369_1_M_I_RB_이상 *)
    R369_1_M_I_RB_자동 AT %MW20080.1 : BOOL; (* R369_1_M_I_RB_자동 *)
    R369_1_M_I_RB_최종작업완료 AT %MW20081.0 : BOOL; (* R369_1_M_I_RB_최종작업완료 *)
    R369_1_M_I_RB_프로그램_이상 AT %MW20080.6 : BOOL; (* R369_1_M_I_RB_프로그램_이상 *)
    R369_1_M_O_RB_1_CYCLE_SET AT %MW21080.3 : BOOL; (* R369_1_M_O_RB_1_CYCLE_SET *)
    R369_1_M_O_RB_1_CYCLE_리셋 AT %MW21080.4 : BOOL; (* R369_1_M_O_RB_1_CYCLE_리셋 *)
    R369_1_M_O_RB_1차_작업완료_리셋 AT %MW21082.0 : BOOL; (* R369_1_M_O_RB_1차_작업완료_리셋 *)
    R369_1_M_O_RB_2차_작업완료_리셋 AT %MW21082.1 : BOOL; (* R369_1_M_O_RB_2차_작업완료_리셋 *)
    R369_1_M_O_RB_2차_진입OK AT %MW21081.8 : BOOL; (* R369_1_M_O_RB_2차_진입OK *)
    R369_1_M_O_RB_3차_작업완료_리셋 AT %MW21082.2 : BOOL; (* R369_1_M_O_RB_3차_작업완료_리셋 *)
    R369_1_M_O_RB_3차_진입OK AT %MW21081.9 : BOOL; (* R369_1_M_O_RB_3차_진입OK *)
    R369_1_M_O_RB_4차_작업완료_리셋 AT %MW21082.3 : BOOL; (* R369_1_M_O_RB_4차_작업완료_리셋 *)
    R369_1_M_O_RB_4차_진입OK AT %MW21081.10 : BOOL; (* R369_1_M_O_RB_4차_진입OK *)
    R369_1_M_O_RB_5차_작업완료_리셋 AT %MW21082.4 : BOOL; (* R369_1_M_O_RB_5차_작업완료_리셋 *)
    R369_1_M_O_RB_5차_진입OK AT %MW21081.11 : BOOL; (* R369_1_M_O_RB_5차_진입OK *)
    R369_1_M_O_RB_6차_작업완료_리셋 AT %MW21082.5 : BOOL; (* R369_1_M_O_RB_6차_작업완료_리셋 *)
    R369_1_M_O_RB_6차_진입OK AT %MW21081.12 : BOOL; (* R369_1_M_O_RB_6차_진입OK *)
    R369_1_M_O_RB_7차_작업완료_리셋 AT %MW21082.6 : BOOL; (* R369_1_M_O_RB_7차_작업완료_리셋 *)
    R369_1_M_O_RB_7차_진입OK AT %MW21081.13 : BOOL; (* R369_1_M_O_RB_7차_진입OK *)
    R369_1_M_O_RB_ATD_OK AT %MW21080.6 : BOOL; (* R369_1_M_O_RB_ATD_OK *)
    R369_1_M_O_RB_PLT_10_진입OK AT %MW21083.10 : BOOL; (* R369_1_M_O_RB_PLT_10_진입OK *)
    R369_1_M_O_RB_PLT_11_진입OK AT %MW21083.11 : BOOL; (* R369_1_M_O_RB_PLT_11_진입OK *)
    R369_1_M_O_RB_PLT_12_진입OK AT %MW21083.12 : BOOL; (* R369_1_M_O_RB_PLT_12_진입OK *)
    R369_1_M_O_RB_PLT_1_진입OK AT %MW21083.1 : BOOL; (* R369_1_M_O_RB_PLT_1_진입OK *)
    R369_1_M_O_RB_PLT_2_진입OK AT %MW21083.2 : BOOL; (* R369_1_M_O_RB_PLT_2_진입OK *)
    R369_1_M_O_RB_PLT_3_진입OK AT %MW21083.3 : BOOL; (* R369_1_M_O_RB_PLT_3_진입OK *)
    R369_1_M_O_RB_PLT_4_진입OK AT %MW21083.4 : BOOL; (* R369_1_M_O_RB_PLT_4_진입OK *)
    R369_1_M_O_RB_PLT_5_진입OK AT %MW21083.5 : BOOL; (* R369_1_M_O_RB_PLT_5_진입OK *)
    R369_1_M_O_RB_PLT_6_진입OK AT %MW21083.6 : BOOL; (* R369_1_M_O_RB_PLT_6_진입OK *)
    R369_1_M_O_RB_PLT_7_진입OK AT %MW21083.7 : BOOL; (* R369_1_M_O_RB_PLT_7_진입OK *)
    R369_1_M_O_RB_PLT_8_진입OK AT %MW21083.8 : BOOL; (* R369_1_M_O_RB_PLT_8_진입OK *)
    R369_1_M_O_RB_PLT_9_진입OK AT %MW21083.9 : BOOL; (* R369_1_M_O_RB_PLT_9_진입OK *)
    R369_1_M_O_RB_PLT_카운터리셋_보조 AT %MW21080.10 : BOOL; (* R369_1_M_O_RB_PLT_카운터리셋_보조 *)
    R369_1_M_O_RB_PROG_NO AT %MW21084 : WORD;
    R369_1_M_O_RB_RESTART_OK AT %MW21080.2 : BOOL; (* R369_1_M_O_RB_RESTART_OK *)
    R369_1_M_O_RB_START_OK AT %MW21080.0 : BOOL; (* R369_1_M_O_RB_START_OK *)
    R369_1_M_O_RB_TEST_MODE_5000회 AT %MW21080.12 : BOOL; (* R369_1_M_O_RB_TEST_MODE_5000회 *)
    R369_1_M_O_RB_TIP_교체_시작 AT %MW21080.7 : BOOL; (* R369_1_M_O_RB_TIP_교체_시작 *)
    R369_1_M_O_RB_TIP_교체_완료 AT %MW21080.8 : BOOL; (* R369_1_M_O_RB_TIP_교체_완료 *)
    R369_1_M_O_RB_VIP_MODE AT %MW21080.11 : BOOL; (* R369_1_M_O_RB_VIP_MODE *)
    R369_1_M_O_RB_냉각수_차단_요청 AT %MW21080.9 : BOOL; (* R369_1_M_O_RB_냉각수_차단_요청 *)
    R369_1_M_O_RB_진입OK_AX차종 AT %MW21081.0 : BOOL; (* R369_1_M_O_RB_진입OK_AX차종 *)
    R369_1_M_O_RB_진입OK_B차종 AT %MW21081.1 : BOOL; (* R369_1_M_O_RB_진입OK_B차종 *)
    R369_1_M_O_RB_진입OK_C차종 AT %MW21081.2 : BOOL; (* R369_1_M_O_RB_진입OK_C차종 *)
    R369_1_M_O_RB_진입OK_D차종 AT %MW21081.3 : BOOL; (* R369_1_M_O_RB_진입OK_D차종 *)
    R369_1_M_O_RB_진입OK_E차종 AT %MW21081.4 : BOOL; (* R369_1_M_O_RB_진입OK_E차종 *)
    R369_1_M_O_RB_진입OK_F차종 AT %MW21081.5 : BOOL; (* R369_1_M_O_RB_진입OK_F차종 *)
    R369_1_M_O_RB_진입OK_G차종 AT %MW21081.6 : BOOL; (* R369_1_M_O_RB_진입OK_G차종 *)
    R369_1_M_O_RB_진입OK_H차종 AT %MW21081.7 : BOOL; (* R369_1_M_O_RB_진입OK_H차종 *)
    R369_1_M_O_RB_최종_작업완료_리셋 AT %MW21080.5 : BOOL; (* R369_1_M_O_RB_최종_작업완료_리셋 *)
    R369_1_M_O_RB_프로그램_OK AT %MW21080.1 : BOOL; (* R369_1_M_O_RB_프로그램_OK *)
    R369_1_O_RB_0_5S_통신_CHK AT %MW94083.14 : BOOL; (* R369_1_O_RB_0_5S_통신_CHK *)
    R369_1_O_RB_2차_진입OK AT %MW94081.8 : BOOL; (* R369_1_O_RB_2차_진입OK *)
    R369_1_O_RB_3차_진입OK AT %MW94081.9 : BOOL; (* R369_1_O_RB_3차_진입OK *)
    R369_1_O_RB_4차_진입OK AT %MW94081.10 : BOOL; (* R369_1_O_RB_4차_진입OK *)
    R369_1_O_RB_5차_진입OK AT %MW94081.11 : BOOL; (* R369_1_O_RB_5차_진입OK *)
    R369_1_O_RB_6차_진입OK AT %MW94081.12 : BOOL; (* R369_1_O_RB_6차_진입OK *)
    R369_1_O_RB_7차_진입OK AT %MW94081.13 : BOOL; (* R369_1_O_RB_7차_진입OK *)
    R369_1_O_RB_AX_1차_진입OK AT %MW94081.0 : BOOL; (* R369_1_O_RB_AX_1차_진입OK *)
    R369_1_O_RB_B_1차_진입OK AT %MW94081.1 : BOOL; (* R369_1_O_RB_B_1차_진입OK *)
    R369_1_O_RB_C_1차_진입OK AT %MW94081.2 : BOOL; (* R369_1_O_RB_C_1차_진입OK *)
    R369_1_O_RB_D_1차_진입OK AT %MW94081.3 : BOOL; (* R369_1_O_RB_D_1차_진입OK *)
    R369_1_O_RB_EACH_작업완료_리셋 AT %MW94080.14 : BOOL; (* R369_1_O_RB_EACH_작업완료_리셋 *)
    R369_1_O_RB_EXT_READY AT %MW94080.11 : BOOL; (* R369_1_O_RB_EXT_READY *)
    R369_1_O_RB_E_1차_진입OK AT %MW94081.4 : BOOL; (* R369_1_O_RB_E_1차_진입OK *)
    R369_1_O_RB_F_1차_진입OK AT %MW94081.5 : BOOL; (* R369_1_O_RB_F_1차_진입OK *)
    R369_1_O_RB_GATE_OPEN_NC AT %MW94083.11 : BOOL; (* R369_1_O_RB_GATE_OPEN_NC *)
    R369_1_O_RB_G_1차_진입OK AT %MW94081.6 : BOOL; (* R369_1_O_RB_G_1차_진입OK *)
    R369_1_O_RB_H_1차_진입OK AT %MW94081.7 : BOOL; (* R369_1_O_RB_H_1차_진입OK *)
    R369_1_O_RB_OUTPUT AT %MW94080 : ARRAY[0..3] OF WORD; (* R369_1_O_RB_OUTPUT *)
    R369_1_O_RB_PAUSE_NC AT %MW94080.13 : BOOL; (* R369_1_O_RB_PAUSE_NC *)
    R369_1_O_RB_PLT10_진입OK AT %MW94082.9 : BOOL; (* R369_1_O_RB_PLT10_진입OK *)
    R369_1_O_RB_PLT11_진입OK AT %MW94082.10 : BOOL; (* R369_1_O_RB_PLT11_진입OK *)
    R369_1_O_RB_PLT12_진입OK AT %MW94082.11 : BOOL; (* R369_1_O_RB_PLT12_진입OK *)
    R369_1_O_RB_PLT1_진입OK AT %MW94082.0 : BOOL; (* R369_1_O_RB_PLT1_진입OK *)
    R369_1_O_RB_PLT2_진입OK AT %MW94082.1 : BOOL; (* R369_1_O_RB_PLT2_진입OK *)
    R369_1_O_RB_PLT3_진입OK AT %MW94082.2 : BOOL; (* R369_1_O_RB_PLT3_진입OK *)
    R369_1_O_RB_PLT4_진입OK AT %MW94082.3 : BOOL; (* R369_1_O_RB_PLT4_진입OK *)
    R369_1_O_RB_PLT5_진입OK AT %MW94082.4 : BOOL; (* R369_1_O_RB_PLT5_진입OK *)
    R369_1_O_RB_PLT6_진입OK AT %MW94082.5 : BOOL; (* R369_1_O_RB_PLT6_진입OK *)
    R369_1_O_RB_PLT7_진입OK AT %MW94082.6 : BOOL; (* R369_1_O_RB_PLT7_진입OK *)
    R369_1_O_RB_PLT8_진입OK AT %MW94082.7 : BOOL; (* R369_1_O_RB_PLT8_진입OK *)
    R369_1_O_RB_PLT9_진입OK AT %MW94082.8 : BOOL; (* R369_1_O_RB_PLT9_진입OK *)
    R369_1_O_RB_PLT_카운터_리셋_요구 AT %MW94083.10 : BOOL; (* R369_1_O_RB_PLT_카운터_리셋_요구 *)
    R369_1_O_RB_PROG_선택1 AT %MW94080.0 : BOOL; (* R369_1_O_RB_PROG_선택1 *)
    R369_1_O_RB_PROG_선택128 AT %MW94080.7 : BOOL; (* R369_1_O_RB_PROG_선택128 *)
    R369_1_O_RB_PROG_선택16 AT %MW94080.4 : BOOL; (* R369_1_O_RB_PROG_선택16 *)
    R369_1_O_RB_PROG_선택2 AT %MW94080.1 : BOOL; (* R369_1_O_RB_PROG_선택2 *)
    R369_1_O_RB_PROG_선택32 AT %MW94080.5 : BOOL; (* R369_1_O_RB_PROG_선택32 *)
    R369_1_O_RB_PROG_선택4 AT %MW94080.2 : BOOL; (* R369_1_O_RB_PROG_선택4 *)
    R369_1_O_RB_PROG_선택64 AT %MW94080.6 : BOOL; (* R369_1_O_RB_PROG_선택64 *)
    R369_1_O_RB_PROG_선택8 AT %MW94080.3 : BOOL; (* R369_1_O_RB_PROG_선택8 *)
    R369_1_O_RB_SP_1_14 AT %MW94081.14 : BOOL; (* R369_1_O_RB_SP_1_14 *)
    R369_1_O_RB_SP_1_15 AT %MW94081.15 : BOOL; (* R369_1_O_RB_SP_1_15 *)
    R369_1_O_RB_SP_2_12 AT %MW94082.12 : BOOL; (* R369_1_O_RB_SP_2_12 *)
    R369_1_O_RB_SP_2_13 AT %MW94082.13 : BOOL; (* R369_1_O_RB_SP_2_13 *)
    R369_1_O_RB_SP_2_14 AT %MW94082.14 : BOOL; (* R369_1_O_RB_SP_2_14 *)
    R369_1_O_RB_SP_5000TH_ON AT %MW94082.15 : BOOL; (* R369_1_O_RB_SP_5000TH_ON *)
    R369_1_O_RB_TIP_CHANGE_END AT %MW94083.9 : BOOL; (* R369_1_O_RB_TIP_CHANGE_END *)
    R369_1_O_RB_TIP_CHANGE_START AT %MW94083.8 : BOOL; (* R369_1_O_RB_TIP_CHANGE_START *)
    R369_1_O_RB_TIP_DRESS_SATRT AT %MW94080.12 : BOOL; (* R369_1_O_RB_TIP_DRESS_SATRT *)
    R369_1_O_RB_VIP_MODE AT %MW94083.15 : BOOL; (* R369_1_O_RB_VIP_MODE *)
    R369_1_O_RB_기동 AT %MW94080.9 : BOOL; (* R369_1_O_RB_기동 *)
    R369_1_O_RB_냉각수차단 AT %MW94080.15 : BOOL; (* R369_1_O_RB_냉각수차단 *)
    R369_1_O_RB_부저정지 AT %MW94083.13 : BOOL; (* R369_1_O_RB_부저정지 *)
    R369_1_O_RB_비상정지_NC AT %MW94083.12 : BOOL; (* R369_1_O_RB_비상정지_NC *)
    R369_1_O_RB_상호인터록_INT1 AT %MW94083.0 : BOOL; (* R369_1_O_RB_상호인터록_INT1 *)
    R369_1_O_RB_상호인터록_INT2 AT %MW94083.1 : BOOL; (* R369_1_O_RB_상호인터록_INT2 *)
    R369_1_O_RB_상호인터록_INT3 AT %MW94083.2 : BOOL; (* R369_1_O_RB_상호인터록_INT3 *)
    R369_1_O_RB_상호인터록_INT4 AT %MW94083.3 : BOOL; (* R369_1_O_RB_상호인터록_INT4 *)
    R369_1_O_RB_상호인터록_INT5 AT %MW94083.4 : BOOL; (* R369_1_O_RB_상호인터록_INT5 *)
    R369_1_O_RB_상호인터록_INT6 AT %MW94083.5 : BOOL; (* R369_1_O_RB_상호인터록_INT6 *)
    R369_1_O_RB_상호인터록_INT7 AT %MW94083.6 : BOOL; (* R369_1_O_RB_상호인터록_INT7 *)
    R369_1_O_RB_상호인터록_INT8 AT %MW94083.7 : BOOL; (* R369_1_O_RB_상호인터록_INT8 *)
    R369_1_O_RB_이상_리셋 AT %MW94080.10 : BOOL; (* R369_1_O_RB_이상_리셋 *)
    R369_1_O_RB_작업완료_리셋 AT %MW94080.8 : BOOL; (* R369_1_O_RB_작업완료_리셋 *)
    R369_2_I_RB_0_5_COMM_CHK AT %MW84093.14 : BOOL; (* R369_2_I_RB_0_5_COMM_CHK *)
    R369_2_I_RB_10차_간섭무 AT %MW84091.9 : BOOL; (* R369_2_I_RB_10차_간섭무 *)
    R369_2_I_RB_11차_간섭무 AT %MW84091.10 : BOOL; (* R369_2_I_RB_11차_간섭무 *)
    R369_2_I_RB_12차_간섭무 AT %MW84091.11 : BOOL; (* R369_2_I_RB_12차_간섭무 *)
    R369_2_I_RB_1차_간섭무 AT %MW84091.0 : BOOL; (* R369_2_I_RB_1차_간섭무 *)
    R369_2_I_RB_1차_작업완료 AT %MW84090.9 : BOOL; (* R369_2_I_RB_1차_작업완료 *)
    R369_2_I_RB_2차_간섭무 AT %MW84091.1 : BOOL; (* R369_2_I_RB_2차_간섭무 *)
    R369_2_I_RB_2차_작업완료 AT %MW84090.10 : BOOL; (* R369_2_I_RB_2차_작업완료 *)
    R369_2_I_RB_3차_간섭무 AT %MW84091.2 : BOOL; (* R369_2_I_RB_3차_간섭무 *)
    R369_2_I_RB_3차_작업완료 AT %MW84090.11 : BOOL; (* R369_2_I_RB_3차_작업완료 *)
    R369_2_I_RB_4차_간섭무 AT %MW84091.3 : BOOL; (* R369_2_I_RB_4차_간섭무 *)
    R369_2_I_RB_4차_작업완료 AT %MW84090.12 : BOOL; (* R369_2_I_RB_4차_작업완료 *)
    R369_2_I_RB_5차_간섭무 AT %MW84091.4 : BOOL; (* R369_2_I_RB_5차_간섭무 *)
    R369_2_I_RB_5차_작업완료 AT %MW84090.13 : BOOL; (* R369_2_I_RB_5차_작업완료 *)
    R369_2_I_RB_6차_간섭무 AT %MW84091.5 : BOOL; (* R369_2_I_RB_6차_간섭무 *)
    R369_2_I_RB_6차_작업완료 AT %MW84090.14 : BOOL; (* R369_2_I_RB_6차_작업완료 *)
    R369_2_I_RB_7차_간섭무 AT %MW84091.6 : BOOL; (* R369_2_I_RB_7차_간섭무 *)
    R369_2_I_RB_7차_작업완료 AT %MW84090.15 : BOOL; (* R369_2_I_RB_7차_작업완료 *)
    R369_2_I_RB_8차_간섭무 AT %MW84091.7 : BOOL; (* R369_2_I_RB_8차_간섭무 *)
    R369_2_I_RB_9차_간섭무 AT %MW84091.8 : BOOL; (* R369_2_I_RB_9차_간섭무 *)
    R369_2_I_RB_AB_NORMAL_선택 AT %MW84090.6 : BOOL; (* R369_2_I_RB_AB_NORMAL_선택 *)
    R369_2_I_RB_GUN1_FIXED_TIP AT %MW84097 : WORD; (* R369_2_I_RB_GUN1_FIXED_TIP *)
    R369_2_I_RB_GUN1_MOVING_TIP AT %MW84096 : WORD; (* R369_2_I_RB_GUN1_MOVING_TIP *)
    R369_2_I_RB_GUN2_FIXED_TIP AT %MW84099 : WORD; (* R369_2_I_RB_GUN2_FIXED_TIP *)
    R369_2_I_RB_GUN2_MOVING_TIP AT %MW84098 : WORD; (* R369_2_I_RB_GUN2_MOVING_TIP *)
    R369_2_I_RB_INPUT AT %MW84090 : ARRAY[0..3] OF WORD; (* R369_2_I_RB_INPUT *)
    R369_2_I_RB_LS_이상 AT %MW84092.11 : BOOL; (* R369_2_I_RB_LS_이상 *)
    R369_2_I_RB_MOTOR_MC_ON AT %MW84093.15 : BOOL; (* R369_2_I_RB_MOTOR_MC_ON *)
    R369_2_I_RB_PLT_UNLOAD_완료 AT %MW84093.11 : BOOL; (* R369_2_I_RB_PLT_UNLOAD_완료 *)
    R369_2_I_RB_PLT_최종UNLOAD_완료 AT %MW84093.12 : BOOL; (* R369_2_I_RB_PLT_최종UNLOAD_완료 *)
    R369_2_I_RB_PROG_ECHO_1 AT %MW84092.0 : BOOL; (* R369_2_I_RB_PROG_ECHO_1 *)
    R369_2_I_RB_PROG_ECHO_128 AT %MW84092.7 : BOOL; (* R369_2_I_RB_PROG_ECHO_128 *)
    R369_2_I_RB_PROG_ECHO_16 AT %MW84092.4 : BOOL; (* R369_2_I_RB_PROG_ECHO_16 *)
    R369_2_I_RB_PROG_ECHO_2 AT %MW84092.1 : BOOL; (* R369_2_I_RB_PROG_ECHO_2 *)
    R369_2_I_RB_PROG_ECHO_32 AT %MW84092.5 : BOOL; (* R369_2_I_RB_PROG_ECHO_32 *)
    R369_2_I_RB_PROG_ECHO_4 AT %MW84092.2 : BOOL; (* R369_2_I_RB_PROG_ECHO_4 *)
    R369_2_I_RB_PROG_ECHO_64 AT %MW84092.6 : BOOL; (* R369_2_I_RB_PROG_ECHO_64 *)
    R369_2_I_RB_PROG_ECHO_8 AT %MW84092.3 : BOOL; (* R369_2_I_RB_PROG_ECHO_8 *)
    R369_2_I_RB_SP3_8 AT %MW84093.8 : BOOL; (* R369_2_I_RB_SP3_8 *)
    R369_2_I_RB_SP3_9 AT %MW84093.9 : BOOL; (* R369_2_I_RB_SP3_9 *)
    R369_2_I_RB_SPARE_WORD_4 AT %MW84094 : WORD; (* R369_2_I_RB_SPARE_WORD_4 *)
    R369_2_I_RB_SP_1_12 AT %MW84091.12 : BOOL; (* R369_2_I_RB_SP_1_12 *)
    R369_2_I_RB_SP_1_13 AT %MW84091.13 : BOOL; (* R369_2_I_RB_SP_1_13 *)
